gfCNCPoint3[7270] = {X 314.6892, Y 8.8093, Z -3.8333, A 0.000, B 0.000, C 0.000 }
gfCNCPoint3[7271] = {X 315.3732, Y 9.4933, Z -3.8333, A 0.000, B 0.000, C 0.000 }
gfCNCPoint3[7272] = {X 315.8879, Y 10.3124, Z -3.8333, A 0.000, B 0.000, C 0.000 }
gfCNCPoint3[7273] = {X 316.2074, Y 11.2255, Z -3.8333, A 0.000, B 0.000, C 0.000 }
gfCNCPoint3[7274] = {X 316.3157, Y 12.1868, Z -3.8333, A 0.000, B 0.000, C 0.000 }
gfCNCPoint3[7275] = {X 316.3157, Y 12.9781, Z -3.8333, A 0.000, B 0.000, C 0.000 }
gfCNCPoint3[7276] = {X 316.2144, Y 13.9082, Z -3.8333, A 0.000, B 0.000, C 0.000 }
gfCNCPoint3[7277] = {X 315.9152, Y 14.7946, Z -3.8333, A 0.000, B 0.000, C 0.000 }
gfCNCPoint3[7278] = {X 315.4322, Y 15.5958, Z -3.8333, A 0.000, B 0.000, C 0.000 }
gfCNCPoint3[7279] = {X 314.7880, Y 16.2743, Z -3.8333, A 0.000, B 0.000, C 0.000 }
gfCNCPoint3[7280] = {X 314.7878, Y 40.9123, Z -3.8333, A 0.000, B 0.000, C 0.000 }
gfCNCPoint3[7281] = {X 315.4264, Y 41.5834, Z -3.8333, A 0.000, B 0.000, C 0.000 }
gfCNCPoint3[7282] = {X 315.9072, Y 42.3751, Z -3.8333, A 0.000, B 0.000, C 0.000 }
gfCNCPoint3[7283] = {X 316.2082, Y 43.2512, Z -3.8333, A 0.000, B 0.000, C 0.000 }
gfCNCPoint3[7284] = {X 316.3156, Y 44.1713, Z -3.8333, A 0.000, B 0.000, C 0.000 }
gfCNCPoint3[7285] = {X 316.3157, Y 45.0000, Z -3.8333, A 0.000, B 0.000, C 0.000 }
gfCNCPoint3[7286] = {X 316.2074, Y 45.9613, Z -3.8333, A 0.000, B 0.000, C 0.000 }
gfCNCPoint3[7287] = {X 315.8879, Y 46.8744, Z -3.8333, A 0.000, B 0.000, C 0.000 }
gfCNCPoint3[7288] = {X 315.3732, Y 47.6935, Z -3.8333, A 0.000, B 0.000, C 0.000 }
gfCNCPoint3[7289] = {X 314.6892, Y 48.3775, Z -3.8333, A 0.000, B 0.000, C 0.000 }
gfCNCPoint3[7290] = {X 313.8701, Y 48.8922, Z -3.8333, A 0.000, B 0.000, C 0.000 }
gfCNCPoint3[7291] = {X 312.9570, Y 49.2117, Z -3.8333, A 0.000, B 0.000, C 0.000 }
gfCNCPoint3[7292] = {X 311.9957, Y 49.3200, Z -3.8333, A 0.000, B 0.000, C 0.000 }
gfCNCPoint3[7293] = {X 305.5523, Y 49.3200, Z -3.8333, A 0.000, B 0.000, C 0.000 }
gfCNCPoint3[7294] = {X 304.5958, Y 49.2128, Z -3.8333, A 0.000, B 0.000, C 0.000 }
gfCNCPoint3[7295] = {X 303.6868, Y 48.8965, Z -3.8333, A 0.000, B 0.000, C 0.000 }
gfCNCPoint3[7296] = {X 302.8704, Y 48.3868, Z -3.8333, A 0.000, B 0.000, C 0.000 }
gfCNCPoint3[7297] = {X 302.1872, Y 47.7090, Z -3.8333, A 0.000, B 0.000, C 0.000 }
gfCNCPoint3[7298] = {X 301.6709, Y 46.8967, Z -3.8333, A 0.000, B 0.000, C 0.000 }
gfCNCPoint3[7299] = {X 301.3473, Y 45.9903, Z -3.8333, A 0.000, B 0.000, C 0.000 }
gfCNCPoint3[7300] = {X 301.2324, Y 45.0348, Z -3.8333, A 0.000, B 0.000, C 0.000 }
gfCNCPoint3[7301] = {X 301.2323, Y 44.2012, Z -3.8333, A 0.000, B 0.000, C 0.000 }
gfCNCPoint3[7302] = {X 301.3501, Y 43.2651, Z -3.8333, A 0.000, B 0.000, C 0.000 }
gfCNCPoint3[7303] = {X 301.6534, Y 42.3717, Z -3.8333, A 0.000, B 0.000, C 0.000 }
gfCNCPoint3[7304] = {X 302.1298, Y 41.5574, Z -3.8333, A 0.000, B 0.000, C 0.000 }
gfCNCPoint3[7305] = {X 302.7601, Y 40.8554, Z -3.8333, A 0.000, B 0.000, C 0.000 }
gfCNCPoint3[7306] = {X 302.7601, Y 34.0343, Z -3.8333, A 0.000, B 0.000, C 0.000 }
gfCNCPoint3[7307] = {X 293.8542, Y 34.0343, Z -3.8333, A 0.000, B 0.000, C 0.000 }
gfCNCPoint3[7308] = {X 293.8534, Y 40.9025, Z -3.8333, A 0.000, B 0.000, C 0.000 }
gfCNCPoint3[7309] = {X 294.4924, Y 41.5865, Z -3.8333, A 0.000, B 0.000, C 0.000 }
gfCNCPoint3[7310] = {X 294.9731, Y 42.3897, Z -3.8333, A 0.000, B 0.000, C 0.000 }
gfCNCPoint3[7311] = {X 295.2739, Y 43.2762, Z -3.8333, A 0.000, B 0.000, C 0.000 }
gfCNCPoint3[7312] = {X 295.3811, Y 44.2061, Z -3.8333, A 0.000, B 0.000, C 0.000 }
gfCNCPoint3[7313] = {X 295.3811, Y 45.0000, Z -3.8333, A 0.000, B 0.000, C 0.000 }
gfCNCPoint3[7314] = {X 295.2728, Y 45.9613, Z -3.8333, A 0.000, B 0.000, C 0.000 }
gfCNCPoint3[7315] = {X 294.9533, Y 46.8744, Z -3.8333, A 0.000, B 0.000, C 0.000 }
gfCNCPoint3[7316] = {X 294.4386, Y 47.6935, Z -3.8333, A 0.000, B 0.000, C 0.000 }
gfCNCPoint3[7317] = {X 293.7546, Y 48.3775, Z -3.8333, A 0.000, B 0.000, C 0.000 }
gfCNCPoint3[7318] = {X 292.9355, Y 48.8922, Z -3.8333, A 0.000, B 0.000, C 0.000 }
gfCNCPoint3[7319] = {X 292.0224, Y 49.2117, Z -3.8333, A 0.000, B 0.000, C 0.000 }
gfCNCPoint3[7320] = {X 291.0611, Y 49.3200, Z -3.8333, A 0.000, B 0.000, C 0.000 }
gfCNCPoint3[7321] = {X 284.6177, Y 49.3200, Z -3.8333, A 0.000, B 0.000, C 0.000 }
gfCNCPoint3[7322] = {X 283.6613, Y 49.2128, Z -3.8333, A 0.000, B 0.000, C 0.000 }
gfCNCPoint3[7323] = {X 282.7524, Y 48.8965, Z -3.8333, A 0.000, B 0.000, C 0.000 }
gfCNCPoint3[7324] = {X 281.9360, Y 48.3869, Z -3.8333, A 0.000, B 0.000, C 0.000 }
gfCNCPoint3[7325] = {X 281.2527, Y 47.7092, Z -3.8333, A 0.000, B 0.000, C 0.000 }
gfCNCPoint3[7326] = {X 280.7365, Y 46.8970, Z -3.8333, A 0.000, B 0.000, C 0.000 }
gfCNCPoint3[7327] = {X 280.4128, Y 45.9907, Z -3.8333, A 0.000, B 0.000, C 0.000 }
gfCNCPoint3[7328] = {X 280.2978, Y 45.0352, Z -3.8333, A 0.000, B 0.000, C 0.000 }
gfCNCPoint3[7329] = {X 280.2977, Y 44.2072, Z -3.8333, A 0.000, B 0.000, C 0.000 }
gfCNCPoint3[7330] = {X 280.4027, Y 43.2782, Z -3.8333, A 0.000, B 0.000, C 0.000 }
gfCNCPoint3[7331] = {X 280.7029, Y 42.3928, Z -3.8333, A 0.000, B 0.000, C 0.000 }
gfCNCPoint3[7332] = {X 281.1846, Y 41.5915, Z -3.8333, A 0.000, B 0.000, C 0.000 }
gfCNCPoint3[7333] = {X 281.8256, Y 40.9110, Z -3.8333, A 0.000, B 0.000, C 0.000 }
gfCNCPoint3[7334] = {X 281.8254, Y 28.5926, Z -3.8333, A 0.000, B 0.000, C 0.000 }
gfCNCPoint3[7335] = {X 277.8254, Y 28.5927, Z -3.8333, A 0.000, B 0.000, C 0.000 }
gfCNCPoint3[7336] = {X 281.9054, Y 28.5926, Z -3.8333, A 0.000, B 0.000, C 0.000 }
gfCNCPoint3[7337] = {X 281.9052, Y 16.2369, Z -3.8333, A 0.000, B 0.000, C 0.000 }
gfCNCPoint3[7338] = {X 281.2671, Y 15.5764, Z -3.8333, A 0.000, B 0.000, C 0.000 }
gfCNCPoint3[7339] = {X 280.7863, Y 14.7940, Z -3.8333, A 0.000, B 0.000, C 0.000 }
gfCNCPoint3[7340] = {X 280.4851, Y 13.9265, Z -3.8333, A 0.000, B 0.000, C 0.000 }
gfCNCPoint3[7341] = {X 280.3778, Y 13.0144, Z -3.8333, A 0.000, B 0.000, C 0.000 }
gfCNCPoint3[7342] = {X 280.3777, Y 12.1868, Z -3.8333, A 0.000, B 0.000, C 0.000 }
gfCNCPoint3[7343] = {X 280.4840, Y 11.2433, Z -3.8333, A 0.000, B 0.000, C 0.000 }
gfCNCPoint3[7344] = {X 280.7976, Y 10.3472, Z -3.8333, A 0.000, B 0.000, C 0.000 }
gfCNCPoint3[7345] = {X 281.3027, Y 9.5432, Z -3.8333, A 0.000, B 0.000, C 0.000 }
gfCNCPoint3[7346] = {X 281.9741, Y 8.8719, Z -3.8333, A 0.000, B 0.000, C 0.000 }
gfCNCPoint3[7347] = {X 282.7780, Y 8.3667, Z -3.8333, A 0.000, B 0.000, C 0.000 }
gfCNCPoint3[7348] = {X 283.6742, Y 8.0531, Z -3.8333, A 0.000, B 0.000, C 0.000 }
gfCNCPoint3[7349] = {X 284.6177, Y 7.9468, Z -3.8333, A 0.000, B 0.000, C 0.000 }
gfCNCPoint3[7350] = {X 291.0611, Y 7.9468, Z -3.8333, A 0.000, B 0.000, C 0.000 }
gfCNCPoint3[7351] = {X 292.0046, Y 8.0531, Z -3.8333, A 0.000, B 0.000, C 0.000 }
gfCNCPoint3[7352] = {X 292.9008, Y 8.3667, Z -3.8333, A 0.000, B 0.000, C 0.000 }
gfCNCPoint3[7353] = {X 293.7047, Y 8.8718, Z -3.8333, A 0.000, B 0.000, C 0.000 }
gfCNCPoint3[7354] = {X 294.3761, Y 9.5432, Z -3.8333, A 0.000, B 0.000, C 0.000 }
gfCNCPoint3[7355] = {X 294.8812, Y 10.3471, Z -3.8333, A 0.000, B 0.000, C 0.000 }
gfCNCPoint3[7356] = {X 295.1948, Y 11.2433, Z -3.8333, A 0.000, B 0.000, C 0.000 }
gfCNCPoint3[7357] = {X 295.3011, Y 12.1868, Z -3.8333, A 0.000, B 0.000, C 0.000 }
gfCNCPoint3[7358] = {X 295.3011, Y 12.9781, Z -3.8333, A 0.000, B 0.000, C 0.000 }
gfCNCPoint3[7359] = {X 295.1996, Y 13.8999, Z -3.8333, A 0.000, B 0.000, C 0.000 }
gfCNCPoint3[7360] = {X 294.9001, Y 14.7776, Z -3.8333, A 0.000, B 0.000, C 0.000 }
gfCNCPoint3[7361] = {X 294.4170, Y 15.5691, Z -3.8333, A 0.000, B 0.000, C 0.000 }
gfCNCPoint3[7362] = {X 293.7733, Y 16.2367, Z -3.8333, A 0.000, B 0.000, C 0.000 }
gfCNCPoint3[7363] = {X 293.7745, Y 22.2765, Z -3.8333, A 0.000, B 0.000, C 0.000 }
gfCNCPoint3[7364] = {X 302.8393, Y 22.2765, Z -3.8333, A 0.000, B 0.000, C 0.000 }
gfCNCPoint3[7365] = {X 302.8443, Y 16.2406, Z -3.8333, A 0.000, B 0.000, C 0.000 }
gfCNCPoint3[7366] = {X 302.2046, Y 15.5801, Z -3.8333, A 0.000, B 0.000, C 0.000 }
gfCNCPoint3[7367] = {X 301.7224, Y 14.7973, Z -3.8333, A 0.000, B 0.000, C 0.000 }
gfCNCPoint3[7368] = {X 301.4203, Y 13.9289, Z -3.8333, A 0.000, B 0.000, C 0.000 }
gfCNCPoint3[7369] = {X 301.3124, Y 13.0158, Z -3.8333, A 0.000, B 0.000, C 0.000 }
gfCNCPoint3[7370] = {X 301.3123, Y 12.1868, Z -3.8333, A 0.000, B 0.000, C 0.000 }
gfCNCPoint3[7371] = {X 301.4186, Y 11.2433, Z -3.8333, A 0.000, B 0.000, C 0.000 }
gfCNCPoint3[7372] = {X 301.7321, Y 10.3471, Z -3.8333, A 0.000, B 0.000, C 0.000 }
gfCNCPoint3[7373] = {X 302.2373, Y 9.5432, Z -3.8333, A 0.000, B 0.000, C 0.000 }
gfCNCPoint3[7374] = {X 302.9087, Y 8.8718, Z -3.8333, A 0.000, B 0.000, C 0.000 }
gfCNCPoint3[7375] = {X 303.7126, Y 8.3667, Z -3.8333, A 0.000, B 0.000, C 0.000 }
gfCNCPoint3[7376] = {X 304.6088, Y 8.0531, Z -3.8333, A 0.000, B 0.000, C 0.000 }
gfCNCPoint3[7377] = {X 305.5523, Y 7.9468, Z -3.8333, A 0.000, B 0.000, C 0.000 }
gfCNCPoint3[7378] = {X 311.9957, Y 7.9468, Z -3.8333, A 0.000, B 0.000, C 0.000 }
gfCNCPoint3[7379] = {X 312.9392, Y 8.0531, Z -3.8333, A 0.000, B 0.000, C 0.000 }
gfCNCPoint3[7380] = {X 313.8354, Y 8.3667, Z -3.8333, A 0.000, B 0.000, C 0.000 }
gfCNCPoint3[7381] = {X 314.6393, Y 8.8718, Z -3.8333, A 0.000, B 0.000, C 0.000 }
gfCNCPoint3[7382] = {X 315.3107, Y 9.5432, Z -3.8333, A 0.000, B 0.000, C 0.000 }
gfCNCPoint3[7383] = {X 315.8158, Y 10.3471, Z -3.8333, A 0.000, B 0.000, C 0.000 }
gfCNCPoint3[7384] = {X 316.1294, Y 11.2433, Z -3.8333, A 0.000, B 0.000, C 0.000 }
gfCNCPoint3[7385] = {X 316.2357, Y 12.1868, Z -3.8333, A 0.000, B 0.000, C 0.000 }
gfCNCPoint3[7386] = {X 316.2357, Y 12.9781, Z -3.8333, A 0.000, B 0.000, C 0.000 }
gfCNCPoint3[7387] = {X 316.1343, Y 13.9000, Z -3.8333, A 0.000, B 0.000, C 0.000 }
gfCNCPoint3[7388] = {X 315.8348, Y 14.7777, Z -3.8333, A 0.000, B 0.000, C 0.000 }
gfCNCPoint3[7389] = {X 315.3517, Y 15.5693, Z -3.8333, A 0.000, B 0.000, C 0.000 }
gfCNCPoint3[7390] = {X 314.7080, Y 16.2370, Z -3.8333, A 0.000, B 0.000, C 0.000 }
gfCNCPoint3[7391] = {X 314.7078, Y 40.9508, Z -3.8333, A 0.000, B 0.000, C 0.000 }
gfCNCPoint3[7392] = {X 314.7361, Y 40.9734, Z -3.8333, A 0.000, B 0.000, C 0.000 }
gfCNCPoint3[7393] = {X 315.3629, Y 41.6320, Z -3.8333, A 0.000, B 0.000, C 0.000 }
gfCNCPoint3[7394] = {X 315.8348, Y 42.4091, Z -3.8333, A 0.000, B 0.000, C 0.000 }
gfCNCPoint3[7395] = {X 316.1302, Y 43.2689, Z -3.8333, A 0.000, B 0.000, C 0.000 }
gfCNCPoint3[7396] = {X 316.2356, Y 44.1720, Z -3.8333, A 0.000, B 0.000, C 0.000 }
gfCNCPoint3[7397] = {X 316.2357, Y 45.0000, Z -3.8333, A 0.000, B 0.000, C 0.000 }
gfCNCPoint3[7398] = {X 316.1294, Y 45.9435, Z -3.8333, A 0.000, B 0.000, C 0.000 }
gfCNCPoint3[7399] = {X 315.8158, Y 46.8397, Z -3.8333, A 0.000, B 0.000, C 0.000 }
gfCNCPoint3[7400] = {X 315.3107, Y 47.6436, Z -3.8333, A 0.000, B 0.000, C 0.000 }
gfCNCPoint3[7401] = {X 314.6393, Y 48.3150, Z -3.8333, A 0.000, B 0.000, C 0.000 }
gfCNCPoint3[7402] = {X 313.8354, Y 48.8201, Z -3.8333, A 0.000, B 0.000, C 0.000 }
gfCNCPoint3[7403] = {X 312.9392, Y 49.1337, Z -3.8333, A 0.000, B 0.000, C 0.000 }
gfCNCPoint3[7404] = {X 311.9957, Y 49.2400, Z -3.8333, A 0.000, B 0.000, C 0.000 }
gfCNCPoint3[7405] = {X 305.5523, Y 49.2400, Z -3.8333, A 0.000, B 0.000, C 0.000 }
gfCNCPoint3[7406] = {X 304.6135, Y 49.1348, Z -3.8333, A 0.000, B 0.000, C 0.000 }
gfCNCPoint3[7407] = {X 303.7214, Y 48.8243, Z -3.8333, A 0.000, B 0.000, C 0.000 }
gfCNCPoint3[7408] = {X 302.9201, Y 48.3241, Z -3.8333, A 0.000, B 0.000, C 0.000 }
gfCNCPoint3[7409] = {X 302.2495, Y 47.6588, Z -3.8333, A 0.000, B 0.000, C 0.000 }
gfCNCPoint3[7410] = {X 301.7428, Y 46.8616, Z -3.8333, A 0.000, B 0.000, C 0.000 }
gfCNCPoint3[7411] = {X 301.4252, Y 45.9720, Z -3.8333, A 0.000, B 0.000, C 0.000 }
gfCNCPoint3[7412] = {X 301.3124, Y 45.0341, Z -3.8333, A 0.000, B 0.000, C 0.000 }
gfCNCPoint3[7413] = {X 301.3123, Y 44.2031, Z -3.8333, A 0.000, B 0.000, C 0.000 }
gfCNCPoint3[7414] = {X 301.4301, Y 43.2745, Z -3.8333, A 0.000, B 0.000, C 0.000 }
gfCNCPoint3[7415] = {X 301.7335, Y 42.3890, Z -3.8333, A 0.000, B 0.000, C 0.000 }
gfCNCPoint3[7416] = {X 302.2101, Y 41.5833, Z -3.8333, A 0.000, B 0.000, C 0.000 }
gfCNCPoint3[7417] = {X 302.8401, Y 40.8909, Z -3.8333, A 0.000, B 0.000, C 0.000 }
gfCNCPoint3[7418] = {X 302.8401, Y 33.9543, Z -3.8333, A 0.000, B 0.000, C 0.000 }
gfCNCPoint3[7419] = {X 293.7742, Y 33.9543, Z -3.8333, A 0.000, B 0.000, C 0.000 }
gfCNCPoint3[7420] = {X 293.7734, Y 40.9393, Z -3.8333, A 0.000, B 0.000, C 0.000 }
gfCNCPoint3[7421] = {X 294.4120, Y 41.6128, Z -3.8333, A 0.000, B 0.000, C 0.000 }
gfCNCPoint3[7422] = {X 294.8928, Y 42.4068, Z -3.8333, A 0.000, B 0.000, C 0.000 }
gfCNCPoint3[7423] = {X 295.1938, Y 43.2848, Z -3.8333, A 0.000, B 0.000, C 0.000 }
gfCNCPoint3[7424] = {X 295.3011, Y 44.2068, Z -3.8333, A 0.000, B 0.000, C 0.000 }
gfCNCPoint3[7425] = {X 295.3011, Y 45.0000, Z -3.8333, A 0.000, B 0.000, C 0.000 }
gfCNCPoint3[7426] = {X 295.1948, Y 45.9435, Z -3.8333, A 0.000, B 0.000, C 0.000 }
gfCNCPoint3[7427] = {X 294.8812, Y 46.8397, Z -3.8333, A 0.000, B 0.000, C 0.000 }
gfCNCPoint3[7428] = {X 294.3761, Y 47.6436, Z -3.8333, A 0.000, B 0.000, C 0.000 }
gfCNCPoint3[7429] = {X 293.7047, Y 48.3150, Z -3.8333, A 0.000, B 0.000, C 0.000 }
gfCNCPoint3[7430] = {X 292.9008, Y 48.8201, Z -3.8333, A 0.000, B 0.000, C 0.000 }
gfCNCPoint3[7431] = {X 292.0046, Y 49.1337, Z -3.8333, A 0.000, B 0.000, C 0.000 }
gfCNCPoint3[7432] = {X 291.0611, Y 49.2400, Z -3.8333, A 0.000, B 0.000, C 0.000 }
gfCNCPoint3[7433] = {X 284.6177, Y 49.2400, Z -3.8333, A 0.000, B 0.000, C 0.000 }
gfCNCPoint3[7434] = {X 283.6790, Y 49.1348, Z -3.8333, A 0.000, B 0.000, C 0.000 }
gfCNCPoint3[7435] = {X 282.7869, Y 48.8244, Z -3.8333, A 0.000, B 0.000, C 0.000 }
gfCNCPoint3[7436] = {X 281.9857, Y 48.3242, Z -3.8333, A 0.000, B 0.000, C 0.000 }
gfCNCPoint3[7437] = {X 281.3150, Y 47.6590, Z -3.8333, A 0.000, B 0.000, C 0.000 }
gfCNCPoint3[7438] = {X 280.8083, Y 46.8619, Z -3.8333, A 0.000, B 0.000, C 0.000 }
gfCNCPoint3[7439] = {X 280.4907, Y 45.9723, Z -3.8333, A 0.000, B 0.000, C 0.000 }
gfCNCPoint3[7440] = {X 280.3778, Y 45.0345, Z -3.8333, A 0.000, B 0.000, C 0.000 }
gfCNCPoint3[7441] = {X 280.3777, Y 44.2076, Z -3.8333, A 0.000, B 0.000, C 0.000 }
gfCNCPoint3[7442] = {X 280.4828, Y 43.2867, Z -3.8333, A 0.000, B 0.000, C 0.000 }
gfCNCPoint3[7443] = {X 280.7832, Y 42.4098, Z -3.8333, A 0.000, B 0.000, C 0.000 }
gfCNCPoint3[7444] = {X 281.2650, Y 41.6180, Z -3.8333, A 0.000, B 0.000, C 0.000 }
gfCNCPoint3[7445] = {X 281.9056, Y 40.9481, Z -3.8333, A 0.000, B 0.000, C 0.000 }
gfCNCPoint3[7446] = {X 281.9054, Y 28.5926, Z -3.8333, A 0.000, B 0.000, C 0.000 }
gfCNCPoint3[7447] = {X 277.9054, Y 28.5927, Z -3.8333, A 0.000, B 0.000, C 0.000 }
gfCNCPoint3[7448] = {X 281.9854, Y 28.5926, Z -3.8333, A 0.000, B 0.000, C 0.000 }
gfCNCPoint3[7449] = {X 281.9852, Y 16.1992, Z -3.8333, A 0.000, B 0.000, C 0.000 }
gfCNCPoint3[7450] = {X 281.3476, Y 15.5495, Z -3.8333, A 0.000, B 0.000, C 0.000 }
gfCNCPoint3[7451] = {X 280.8666, Y 14.7766, Z -3.8333, A 0.000, B 0.000, C 0.000 }
gfCNCPoint3[7452] = {X 280.5652, Y 13.9177, Z -3.8333, A 0.000, B 0.000, C 0.000 }
gfCNCPoint3[7453] = {X 280.4578, Y 13.0137, Z -3.8333, A 0.000, B 0.000, C 0.000 }
gfCNCPoint3[7454] = {X 280.4577, Y 12.1868, Z -3.8333, A 0.000, B 0.000, C 0.000 }
gfCNCPoint3[7455] = {X 280.5620, Y 11.2611, Z -3.8333, A 0.000, B 0.000, C 0.000 }
gfCNCPoint3[7456] = {X 280.8696, Y 10.3819, Z -3.8333, A 0.000, B 0.000, C 0.000 }
gfCNCPoint3[7457] = {X 281.3652, Y 9.5931, Z -3.8333, A 0.000, B 0.000, C 0.000 }
gfCNCPoint3[7458] = {X 282.0240, Y 8.9344, Z -3.8333, A 0.000, B 0.000, C 0.000 }
gfCNCPoint3[7459] = {X 282.8127, Y 8.4388, Z -3.8333, A 0.000, B 0.000, C 0.000 }
gfCNCPoint3[7460] = {X 283.6920, Y 8.1311, Z -3.8333, A 0.000, B 0.000, C 0.000 }
gfCNCPoint3[7461] = {X 284.6177, Y 8.0268, Z -3.8333, A 0.000, B 0.000, C 0.000 }
gfCNCPoint3[7462] = {X 291.0611, Y 8.0268, Z -3.8333, A 0.000, B 0.000, C 0.000 }
gfCNCPoint3[7463] = {X 291.9868, Y 8.1311, Z -3.8333, A 0.000, B 0.000, C 0.000 }
gfCNCPoint3[7464] = {X 292.8661, Y 8.4388, Z -3.8333, A 0.000, B 0.000, C 0.000 }
gfCNCPoint3[7465] = {X 293.6549, Y 8.9344, Z -3.8333, A 0.000, B 0.000, C 0.000 }
gfCNCPoint3[7466] = {X 294.3136, Y 9.5931, Z -3.8333, A 0.000, B 0.000, C 0.000 }
gfCNCPoint3[7467] = {X 294.8092, Y 10.3819, Z -3.8333, A 0.000, B 0.000, C 0.000 }
gfCNCPoint3[7468] = {X 295.1168, Y 11.2611, Z -3.8333, A 0.000, B 0.000, C 0.000 }
gfCNCPoint3[7469] = {X 295.2211, Y 12.1868, Z -3.8333, A 0.000, B 0.000, C 0.000 }
gfCNCPoint3[7470] = {X 295.2211, Y 12.9781, Z -3.8333, A 0.000, B 0.000, C 0.000 }
gfCNCPoint3[7471] = {X 295.1254, Y 13.8652, Z -3.8333, A 0.000, B 0.000, C 0.000 }
gfCNCPoint3[7472] = {X 294.8428, Y 14.7115, Z -3.8333, A 0.000, B 0.000, C 0.000 }
gfCNCPoint3[7473] = {X 294.3862, Y 15.4780, Z -3.8333, A 0.000, B 0.000, C 0.000 }
gfCNCPoint3[7474] = {X 293.7766, Y 16.1295, Z -3.8333, A 0.000, B 0.000, C 0.000 }
gfCNCPoint3[7475] = {X 293.6933, Y 16.1994, Z -3.8333, A 0.000, B 0.000, C 0.000 }
gfCNCPoint3[7476] = {X 293.6945, Y 22.3566, Z -3.8333, A 0.000, B 0.000, C 0.000 }
gfCNCPoint3[7477] = {X 302.9192, Y 22.3565, Z -3.8333, A 0.000, B 0.000, C 0.000 }
gfCNCPoint3[7478] = {X 302.9243, Y 16.2028, Z -3.8333, A 0.000, B 0.000, C 0.000 }
gfCNCPoint3[7479] = {X 302.2851, Y 15.5532, Z -3.8333, A 0.000, B 0.000, C 0.000 }
gfCNCPoint3[7480] = {X 301.8027, Y 14.7799, Z -3.8333, A 0.000, B 0.000, C 0.000 }
gfCNCPoint3[7481] = {X 301.5003, Y 13.9201, Z -3.8333, A 0.000, B 0.000, C 0.000 }
gfCNCPoint3[7482] = {X 301.3924, Y 13.0151, Z -3.8333, A 0.000, B 0.000, C 0.000 }
gfCNCPoint3[7483] = {X 301.3923, Y 12.1868, Z -3.8333, A 0.000, B 0.000, C 0.000 }
gfCNCPoint3[7484] = {X 301.4966, Y 11.2611, Z -3.8333, A 0.000, B 0.000, C 0.000 }
gfCNCPoint3[7485] = {X 301.8042, Y 10.3819, Z -3.8333, A 0.000, B 0.000, C 0.000 }
gfCNCPoint3[7486] = {X 302.2998, Y 9.5931, Z -3.8333, A 0.000, B 0.000, C 0.000 }
gfCNCPoint3[7487] = {X 302.9585, Y 8.9344, Z -3.8333, A 0.000, B 0.000, C 0.000 }
gfCNCPoint3[7488] = {X 303.7473, Y 8.4388, Z -3.8333, A 0.000, B 0.000, C 0.000 }
gfCNCPoint3[7489] = {X 304.6266, Y 8.1311, Z -3.8333, A 0.000, B 0.000, C 0.000 }
gfCNCPoint3[7490] = {X 305.5523, Y 8.0268, Z -3.8333, A 0.000, B 0.000, C 0.000 }
gfCNCPoint3[7491] = {X 311.9957, Y 8.0268, Z -3.8333, A 0.000, B 0.000, C 0.000 }
gfCNCPoint3[7492] = {X 312.9214, Y 8.1311, Z -3.8333, A 0.000, B 0.000, C 0.000 }
gfCNCPoint3[7493] = {X 313.8007, Y 8.4388, Z -3.8333, A 0.000, B 0.000, C 0.000 }
gfCNCPoint3[7494] = {X 314.5894, Y 8.9344, Z -3.8333, A 0.000, B 0.000, C 0.000 }
gfCNCPoint3[7495] = {X 315.2481, Y 9.5931, Z -3.8333, A 0.000, B 0.000, C 0.000 }
gfCNCPoint3[7496] = {X 315.7438, Y 10.3819, Z -3.8333, A 0.000, B 0.000, C 0.000 }
gfCNCPoint3[7497] = {X 316.0514, Y 11.2611, Z -3.8333, A 0.000, B 0.000, C 0.000 }
gfCNCPoint3[7498] = {X 316.1557, Y 12.1868, Z -3.8333, A 0.000, B 0.000, C 0.000 }
gfCNCPoint3[7499] = {X 316.1557, Y 12.9781, Z -3.8333, A 0.000, B 0.000, C 0.000 }
gfCNCPoint3[7500] = {X 316.0542, Y 13.8916, Z -3.8333, A 0.000, B 0.000, C 0.000 }
gfCNCPoint3[7501] = {X 315.7545, Y 14.7604, Z -3.8333, A 0.000, B 0.000, C 0.000 }
gfCNCPoint3[7502] = {X 315.2715, Y 15.5422, Z -3.8333, A 0.000, B 0.000, C 0.000 }
gfCNCPoint3[7503] = {X 314.6285, Y 16.1989, Z -3.8333, A 0.000, B 0.000, C 0.000 }
gfCNCPoint3[7504] = {X 314.6278, Y 40.9894, Z -3.8333, A 0.000, B 0.000, C 0.000 }
gfCNCPoint3[7505] = {X 314.6834, Y 41.0336, Z -3.8333, A 0.000, B 0.000, C 0.000 }
gfCNCPoint3[7506] = {X 315.2987, Y 41.6798, Z -3.8333, A 0.000, B 0.000, C 0.000 }
gfCNCPoint3[7507] = {X 315.7621, Y 42.4424, Z -3.8333, A 0.000, B 0.000, C 0.000 }
gfCNCPoint3[7508] = {X 316.0522, Y 43.2863, Z -3.8333, A 0.000, B 0.000, C 0.000 }
gfCNCPoint3[7509] = {X 316.1556, Y 44.1727, Z -3.8333, A 0.000, B 0.000, C 0.000 }
gfCNCPoint3[7510] = {X 316.1557, Y 45.0000, Z -3.8333, A 0.000, B 0.000, C 0.000 }
gfCNCPoint3[7511] = {X 316.0514, Y 45.9257, Z -3.8333, A 0.000, B 0.000, C 0.000 }
gfCNCPoint3[7512] = {X 315.7438, Y 46.8050, Z -3.8333, A 0.000, B 0.000, C 0.000 }
gfCNCPoint3[7513] = {X 315.2481, Y 47.5937, Z -3.8333, A 0.000, B 0.000, C 0.000 }
gfCNCPoint3[7514] = {X 314.5894, Y 48.2524, Z -3.8333, A 0.000, B 0.000, C 0.000 }
gfCNCPoint3[7515] = {X 313.8007, Y 48.7480, Z -3.8333, A 0.000, B 0.000, C 0.000 }
gfCNCPoint3[7516] = {X 312.9214, Y 49.0557, Z -3.8333, A 0.000, B 0.000, C 0.000 }
gfCNCPoint3[7517] = {X 311.9957, Y 49.1600, Z -3.8333, A 0.000, B 0.000, C 0.000 }
gfCNCPoint3[7518] = {X 305.5523, Y 49.1600, Z -3.8333, A 0.000, B 0.000, C 0.000 }
gfCNCPoint3[7519] = {X 304.6312, Y 49.0568, Z -3.8333, A 0.000, B 0.000, C 0.000 }
gfCNCPoint3[7520] = {X 303.7559, Y 48.7522, Z -3.8333, A 0.000, B 0.000, C 0.000 }
gfCNCPoint3[7521] = {X 302.9698, Y 48.2613, Z -3.8333, A 0.000, B 0.000, C 0.000 }
gfCNCPoint3[7522] = {X 302.3118, Y 47.6087, Z -3.8333, A 0.000, B 0.000, C 0.000 }
gfCNCPoint3[7523] = {X 301.8147, Y 46.8265, Z -3.8333, A 0.000, B 0.000, C 0.000 }
gfCNCPoint3[7524] = {X 301.5030, Y 45.9537, Z -3.8333, A 0.000, B 0.000, C 0.000 }
gfCNCPoint3[7525] = {X 301.3924, Y 45.0335, Z -3.8333, A 0.000, B 0.000, C 0.000 }
gfCNCPoint3[7526] = {X 301.3923, Y 44.2050, Z -3.8333, A 0.000, B 0.000, C 0.000 }
gfCNCPoint3[7527] = {X 301.5100, Y 43.2839, Z -3.8333, A 0.000, B 0.000, C 0.000 }
gfCNCPoint3[7528] = {X 301.8136, Y 42.4063, Z -3.8333, A 0.000, B 0.000, C 0.000 }
gfCNCPoint3[7529] = {X 302.2904, Y 41.6094, Z -3.8333, A 0.000, B 0.000, C 0.000 }
gfCNCPoint3[7530] = {X 302.9201, Y 40.9268, Z -3.8333, A 0.000, B 0.000, C 0.000 }
gfCNCPoint3[7531] = {X 302.9201, Y 33.8743, Z -3.8333, A 0.000, B 0.000, C 0.000 }
gfCNCPoint3[7532] = {X 293.6942, Y 33.8743, Z -3.8333, A 0.000, B 0.000, C 0.000 }
gfCNCPoint3[7533] = {X 293.6934, Y 40.9764, Z -3.8333, A 0.000, B 0.000, C 0.000 }
gfCNCPoint3[7534] = {X 294.3316, Y 41.6394, Z -3.8333, A 0.000, B 0.000, C 0.000 }
gfCNCPoint3[7535] = {X 294.8125, Y 42.4240, Z -3.8333, A 0.000, B 0.000, C 0.000 }
gfCNCPoint3[7536] = {X 295.1137, Y 43.2935, Z -3.8333, A 0.000, B 0.000, C 0.000 }
gfCNCPoint3[7537] = {X 295.2211, Y 44.2075, Z -3.8333, A 0.000, B 0.000, C 0.000 }
gfCNCPoint3[7538] = {X 295.2211, Y 45.0000, Z -3.8333, A 0.000, B 0.000, C 0.000 }
gfCNCPoint3[7539] = {X 295.1168, Y 45.9257, Z -3.8333, A 0.000, B 0.000, C 0.000 }
gfCNCPoint3[7540] = {X 294.8092, Y 46.8050, Z -3.8333, A 0.000, B 0.000, C 0.000 }
gfCNCPoint3[7541] = {X 294.3136, Y 47.5937, Z -3.8333, A 0.000, B 0.000, C 0.000 }
gfCNCPoint3[7542] = {X 293.6549, Y 48.2524, Z -3.8333, A 0.000, B 0.000, C 0.000 }
gfCNCPoint3[7543] = {X 292.8661, Y 48.7480, Z -3.8333, A 0.000, B 0.000, C 0.000 }
gfCNCPoint3[7544] = {X 291.9868, Y 49.0557, Z -3.8333, A 0.000, B 0.000, C 0.000 }
gfCNCPoint3[7545] = {X 291.0611, Y 49.1600, Z -3.8333, A 0.000, B 0.000, C 0.000 }
gfCNCPoint3[7546] = {X 284.6177, Y 49.1600, Z -3.8333, A 0.000, B 0.000, C 0.000 }
gfCNCPoint3[7547] = {X 283.6967, Y 49.0568, Z -3.8333, A 0.000, B 0.000, C 0.000 }
gfCNCPoint3[7548] = {X 282.8214, Y 48.7522, Z -3.8333, A 0.000, B 0.000, C 0.000 }
gfCNCPoint3[7549] = {X 282.0353, Y 48.2615, Z -3.8333, A 0.000, B 0.000, C 0.000 }
gfCNCPoint3[7550] = {X 281.3774, Y 47.6088, Z -3.8333, A 0.000, B 0.000, C 0.000 }
gfCNCPoint3[7551] = {X 280.8802, Y 46.8267, Z -3.8333, A 0.000, B 0.000, C 0.000 }
gfCNCPoint3[7552] = {X 280.5685, Y 45.9540, Z -3.8333, A 0.000, B 0.000, C 0.000 }
gfCNCPoint3[7553] = {X 280.4578, Y 45.0339, Z -3.8333, A 0.000, B 0.000, C 0.000 }
gfCNCPoint3[7554] = {X 280.4577, Y 44.2080, Z -3.8333, A 0.000, B 0.000, C 0.000 }
gfCNCPoint3[7555] = {X 280.5629, Y 43.2952, Z -3.8333, A 0.000, B 0.000, C 0.000 }
gfCNCPoint3[7556] = {X 280.8636, Y 42.4270, Z -3.8333, A 0.000, B 0.000, C 0.000 }
gfCNCPoint3[7557] = {X 281.3455, Y 41.6447, Z -3.8333, A 0.000, B 0.000, C 0.000 }
gfCNCPoint3[7558] = {X 281.9856, Y 40.9855, Z -3.8333, A 0.000, B 0.000, C 0.000 }
gfCNCPoint3[7559] = {X 281.9854, Y 28.5926, Z -3.8333, A 0.000, B 0.000, C 0.000 }
gfCNCPoint3[7560] = {X 277.9854, Y 28.5927, Z -3.8333, A 0.000, B 0.000, C 0.000 }
gfCNCPoint3[7561] = {X 282.0654, Y 28.5926, Z -3.8333, A 0.000, B 0.000, C 0.000 }
gfCNCPoint3[7562] = {X 282.0652, Y 16.1610, Z -3.8333, A 0.000, B 0.000, C 0.000 }
gfCNCPoint3[7563] = {X 281.4281, Y 15.5222, Z -3.8333, A 0.000, B 0.000, C 0.000 }
gfCNCPoint3[7564] = {X 280.9469, Y 14.7591, Z -3.8333, A 0.000, B 0.000, C 0.000 }
gfCNCPoint3[7565] = {X 280.6453, Y 13.9088, Z -3.8333, A 0.000, B 0.000, C 0.000 }
gfCNCPoint3[7566] = {X 280.5378, Y 13.0130, Z -3.8333, A 0.000, B 0.000, C 0.000 }
gfCNCPoint3[7567] = {X 280.5377, Y 12.1868, Z -3.8333, A 0.000, B 0.000, C 0.000 }
gfCNCPoint3[7568] = {X 280.6400, Y 11.2789, Z -3.8333, A 0.000, B 0.000, C 0.000 }
gfCNCPoint3[7569] = {X 280.9417, Y 10.4166, Z -3.8333, A 0.000, B 0.000, C 0.000 }
gfCNCPoint3[7570] = {X 281.4278, Y 9.6430, Z -3.8333, A 0.000, B 0.000, C 0.000 }
gfCNCPoint3[7571] = {X 282.0738, Y 8.9969, Z -3.8333, A 0.000, B 0.000, C 0.000 }
gfCNCPoint3[7572] = {X 282.8474, Y 8.5109, Z -3.8333, A 0.000, B 0.000, C 0.000 }
gfCNCPoint3[7573] = {X 283.7098, Y 8.2091, Z -3.8333, A 0.000, B 0.000, C 0.000 }
gfCNCPoint3[7574] = {X 284.6177, Y 8.1068, Z -3.8333, A 0.000, B 0.000, C 0.000 }
gfCNCPoint3[7575] = {X 291.0611, Y 8.1068, Z -3.8333, A 0.000, B 0.000, C 0.000 }
gfCNCPoint3[7576] = {X 291.9690, Y 8.2091, Z -3.8333, A 0.000, B 0.000, C 0.000 }
gfCNCPoint3[7577] = {X 292.8314, Y 8.5109, Z -3.8333, A 0.000, B 0.000, C 0.000 }
gfCNCPoint3[7578] = {X 293.6050, Y 8.9969, Z -3.8333, A 0.000, B 0.000, C 0.000 }
gfCNCPoint3[7579] = {X 294.2510, Y 9.6430, Z -3.8333, A 0.000, B 0.000, C 0.000 }
gfCNCPoint3[7580] = {X 294.7371, Y 10.4166, Z -3.8333, A 0.000, B 0.000, C 0.000 }
gfCNCPoint3[7581] = {X 295.0388, Y 11.2789, Z -3.8333, A 0.000, B 0.000, C 0.000 }
gfCNCPoint3[7582] = {X 295.1411, Y 12.1868, Z -3.8333, A 0.000, B 0.000, C 0.000 }
gfCNCPoint3[7583] = {X 295.1411, Y 12.9781, Z -3.8333, A 0.000, B 0.000, C 0.000 }
gfCNCPoint3[7584] = {X 295.0473, Y 13.8481, Z -3.8333, A 0.000, B 0.000, C 0.000 }
gfCNCPoint3[7585] = {X 294.7701, Y 14.6781, Z -3.8333, A 0.000, B 0.000, C 0.000 }
gfCNCPoint3[7586] = {X 294.3222, Y 15.4299, Z -3.8333, A 0.000, B 0.000, C 0.000 }
gfCNCPoint3[7587] = {X 293.7244, Y 16.0689, Z -3.8333, A 0.000, B 0.000, C 0.000 }
gfCNCPoint3[7588] = {X 293.6670, Y 16.1174, Z -3.8333, A 0.000, B 0.000, C 0.000 }
gfCNCPoint3[7589] = {X 293.6087, Y 16.1649, Z -3.8333, A 0.000, B 0.000, C 0.000 }
gfCNCPoint3[7590] = {X 293.6133, Y 16.1995, Z -3.8333, A 0.000, B 0.000, C 0.000 }
gfCNCPoint3[7591] = {X 293.6145, Y 22.4367, Z -3.8333, A 0.000, B 0.000, C 0.000 }
gfCNCPoint3[7592] = {X 293.7676, Y 22.4365, Z -3.8333, A 0.000, B 0.000, C 0.000 }
gfCNCPoint3[7593] = {X 302.9992, Y 22.4365, Z -3.8333, A 0.000, B 0.000, C 0.000 }
gfCNCPoint3[7594] = {X 303.0043, Y 16.1646, Z -3.8333, A 0.000, B 0.000, C 0.000 }
gfCNCPoint3[7595] = {X 302.9460, Y 16.1171, Z -3.8333, A 0.000, B 0.000, C 0.000 }
gfCNCPoint3[7596] = {X 302.8886, Y 16.0686, Z -3.8333, A 0.000, B 0.000, C 0.000 }
gfCNCPoint3[7597] = {X 302.2964, Y 15.4368, Z -3.8333, A 0.000, B 0.000, C 0.000 }
gfCNCPoint3[7598] = {X 301.8508, Y 14.6944, Z -3.8333, A 0.000, B 0.000, C 0.000 }
gfCNCPoint3[7599] = {X 301.5720, Y 13.8746, Z -3.8333, A 0.000, B 0.000, C 0.000 }
gfCNCPoint3[7600] = {X 301.4724, Y 13.0144, Z -3.8333, A 0.000, B 0.000, C 0.000 }
gfCNCPoint3[7601] = {X 301.4723, Y 12.1868, Z -3.8333, A 0.000, B 0.000, C 0.000 }
gfCNCPoint3[7602] = {X 301.5745, Y 11.2789, Z -3.8333, A 0.000, B 0.000, C 0.000 }
gfCNCPoint3[7603] = {X 301.8763, Y 10.4166, Z -3.8333, A 0.000, B 0.000, C 0.000 }
gfCNCPoint3[7604] = {X 302.3624, Y 9.6430, Z -3.8333, A 0.000, B 0.000, C 0.000 }
gfCNCPoint3[7605] = {X 303.0084, Y 8.9969, Z -3.8333, A 0.000, B 0.000, C 0.000 }
gfCNCPoint3[7606] = {X 303.7820, Y 8.5109, Z -3.8333, A 0.000, B 0.000, C 0.000 }
gfCNCPoint3[7607] = {X 304.6444, Y 8.2091, Z -3.8333, A 0.000, B 0.000, C 0.000 }
gfCNCPoint3[7608] = {X 305.5523, Y 8.1068, Z -3.8333, A 0.000, B 0.000, C 0.000 }
gfCNCPoint3[7609] = {X 311.9957, Y 8.1068, Z -3.8333, A 0.000, B 0.000, C 0.000 }
gfCNCPoint3[7610] = {X 312.9036, Y 8.2091, Z -3.8333, A 0.000, B 0.000, C 0.000 }
gfCNCPoint3[7611] = {X 313.7660, Y 8.5109, Z -3.8333, A 0.000, B 0.000, C 0.000 }
gfCNCPoint3[7612] = {X 314.5396, Y 8.9969, Z -3.8333, A 0.000, B 0.000, C 0.000 }
gfCNCPoint3[7613] = {X 315.1856, Y 9.6430, Z -3.8333, A 0.000, B 0.000, C 0.000 }
gfCNCPoint3[7614] = {X 315.6717, Y 10.4166, Z -3.8333, A 0.000, B 0.000, C 0.000 }
gfCNCPoint3[7615] = {X 315.9734, Y 11.2789, Z -3.8333, A 0.000, B 0.000, C 0.000 }
gfCNCPoint3[7616] = {X 316.0757, Y 12.1868, Z -3.8333, A 0.000, B 0.000, C 0.000 }
gfCNCPoint3[7617] = {X 316.0757, Y 12.9781, Z -3.8333, A 0.000, B 0.000, C 0.000 }
gfCNCPoint3[7618] = {X 315.9819, Y 13.8481, Z -3.8333, A 0.000, B 0.000, C 0.000 }
gfCNCPoint3[7619] = {X 315.7047, Y 14.6780, Z -3.8333, A 0.000, B 0.000, C 0.000 }
gfCNCPoint3[7620] = {X 315.2569, Y 15.4298, Z -3.8333, A 0.000, B 0.000, C 0.000 }
gfCNCPoint3[7621] = {X 314.6591, Y 16.0687, Z -3.8333, A 0.000, B 0.000, C 0.000 }
gfCNCPoint3[7622] = {X 314.6045, Y 16.1150, Z -3.8333, A 0.000, B 0.000, C 0.000 }
gfCNCPoint3[7623] = {X 314.5490, Y 16.1603, Z -3.8333, A 0.000, B 0.000, C 0.000 }
gfCNCPoint3[7624] = {X 314.5478, Y 41.0280, Z -3.8333, A 0.000, B 0.000, C 0.000 }
gfCNCPoint3[7625] = {X 314.6336, Y 41.0962, Z -3.8333, A 0.000, B 0.000, C 0.000 }
gfCNCPoint3[7626] = {X 315.2363, Y 41.7299, Z -3.8333, A 0.000, B 0.000, C 0.000 }
gfCNCPoint3[7627] = {X 315.6902, Y 42.4775, Z -3.8333, A 0.000, B 0.000, C 0.000 }
gfCNCPoint3[7628] = {X 315.9743, Y 43.3047, Z -3.8333, A 0.000, B 0.000, C 0.000 }
gfCNCPoint3[7629] = {X 316.0756, Y 44.1734, Z -3.8333, A 0.000, B 0.000, C 0.000 }
gfCNCPoint3[7630] = {X 316.0757, Y 45.0000, Z -3.8333, A 0.000, B 0.000, C 0.000 }
gfCNCPoint3[7631] = {X 315.9734, Y 45.9079, Z -3.8333, A 0.000, B 0.000, C 0.000 }
gfCNCPoint3[7632] = {X 315.6717, Y 46.7702, Z -3.8333, A 0.000, B 0.000, C 0.000 }
gfCNCPoint3[7633] = {X 315.1856, Y 47.5438, Z -3.8333, A 0.000, B 0.000, C 0.000 }
gfCNCPoint3[7634] = {X 314.5396, Y 48.1899, Z -3.8333, A 0.000, B 0.000, C 0.000 }
gfCNCPoint3[7635] = {X 313.7660, Y 48.6760, Z -3.8333, A 0.000, B 0.000, C 0.000 }
gfCNCPoint3[7636] = {X 312.9036, Y 48.9777, Z -3.8333, A 0.000, B 0.000, C 0.000 }
gfCNCPoint3[7637] = {X 311.9957, Y 49.0800, Z -3.8333, A 0.000, B 0.000, C 0.000 }
gfCNCPoint3[7638] = {X 305.5523, Y 49.0800, Z -3.8333, A 0.000, B 0.000, C 0.000 }
gfCNCPoint3[7639] = {X 304.6489, Y 48.9787, Z -3.8333, A 0.000, B 0.000, C 0.000 }
gfCNCPoint3[7640] = {X 303.7905, Y 48.6800, Z -3.8333, A 0.000, B 0.000, C 0.000 }
gfCNCPoint3[7641] = {X 303.0194, Y 48.1986, Z -3.8333, A 0.000, B 0.000, C 0.000 }
gfCNCPoint3[7642] = {X 302.3741, Y 47.5585, Z -3.8333, A 0.000, B 0.000, C 0.000 }
gfCNCPoint3[7643] = {X 301.8865, Y 46.7914, Z -3.8333, A 0.000, B 0.000, C 0.000 }
gfCNCPoint3[7644] = {X 301.5809, Y 45.9353, Z -3.8333, A 0.000, B 0.000, C 0.000 }
gfCNCPoint3[7645] = {X 301.4724, Y 45.0328, Z -3.8333, A 0.000, B 0.000, C 0.000 }
gfCNCPoint3[7646] = {X 301.4723, Y 44.2070, Z -3.8333, A 0.000, B 0.000, C 0.000 }
gfCNCPoint3[7647] = {X 301.5900, Y 43.2934, Z -3.8333, A 0.000, B 0.000, C 0.000 }
gfCNCPoint3[7648] = {X 301.8938, Y 42.4238, Z -3.8333, A 0.000, B 0.000, C 0.000 }
gfCNCPoint3[7649] = {X 302.3707, Y 41.6357, Z -3.8333, A 0.000, B 0.000, C 0.000 }
gfCNCPoint3[7650] = {X 303.0001, Y 40.9632, Z -3.8333, A 0.000, B 0.000, C 0.000 }
gfCNCPoint3[7651] = {X 303.0001, Y 33.7943, Z -3.8333, A 0.000, B 0.000, C 0.000 }
gfCNCPoint3[7652] = {X 293.6143, Y 33.7943, Z -3.8333, A 0.000, B 0.000, C 0.000 }
gfCNCPoint3[7653] = {X 293.6134, Y 41.0141, Z -3.8333, A 0.000, B 0.000, C 0.000 }
gfCNCPoint3[7654] = {X 294.2511, Y 41.6663, Z -3.8333, A 0.000, B 0.000, C 0.000 }
gfCNCPoint3[7655] = {X 294.7322, Y 42.4413, Z -3.8333, A 0.000, B 0.000, C 0.000 }
gfCNCPoint3[7656] = {X 295.0337, Y 43.3023, Z -3.8333, A 0.000, B 0.000, C 0.000 }
gfCNCPoint3[7657] = {X 295.1411, Y 44.2082, Z -3.8333, A 0.000, B 0.000, C 0.000 }
gfCNCPoint3[7658] = {X 295.1411, Y 45.0000, Z -3.8333, A 0.000, B 0.000, C 0.000 }
gfCNCPoint3[7659] = {X 295.0388, Y 45.9079, Z -3.8333, A 0.000, B 0.000, C 0.000 }
gfCNCPoint3[7660] = {X 294.7371, Y 46.7702, Z -3.8333, A 0.000, B 0.000, C 0.000 }
gfCNCPoint3[7661] = {X 294.2510, Y 47.5438, Z -3.8333, A 0.000, B 0.000, C 0.000 }
gfCNCPoint3[7662] = {X 293.6050, Y 48.1899, Z -3.8333, A 0.000, B 0.000, C 0.000 }
gfCNCPoint3[7663] = {X 292.8314, Y 48.6760, Z -3.8333, A 0.000, B 0.000, C 0.000 }
gfCNCPoint3[7664] = {X 291.9690, Y 48.9777, Z -3.8333, A 0.000, B 0.000, C 0.000 }
gfCNCPoint3[7665] = {X 291.0611, Y 49.0800, Z -3.8333, A 0.000, B 0.000, C 0.000 }
gfCNCPoint3[7666] = {X 284.6177, Y 49.0800, Z -3.8333, A 0.000, B 0.000, C 0.000 }
gfCNCPoint3[7667] = {X 283.7144, Y 48.9788, Z -3.8333, A 0.000, B 0.000, C 0.000 }
gfCNCPoint3[7668] = {X 282.8560, Y 48.6801, Z -3.8333, A 0.000, B 0.000, C 0.000 }
gfCNCPoint3[7669] = {X 282.0850, Y 48.1987, Z -3.8333, A 0.000, B 0.000, C 0.000 }
gfCNCPoint3[7670] = {X 281.4397, Y 47.5587, Z -3.8333, A 0.000, B 0.000, C 0.000 }
gfCNCPoint3[7671] = {X 280.9521, Y 46.7916, Z -3.8333, A 0.000, B 0.000, C 0.000 }
gfCNCPoint3[7672] = {X 280.6464, Y 45.9356, Z -3.8333, A 0.000, B 0.000, C 0.000 }
gfCNCPoint3[7673] = {X 280.5378, Y 45.0332, Z -3.8333, A 0.000, B 0.000, C 0.000 }
gfCNCPoint3[7674] = {X 280.5377, Y 44.2085, Z -3.8333, A 0.000, B 0.000, C 0.000 }
gfCNCPoint3[7675] = {X 280.6430, Y 43.3039, Z -3.8333, A 0.000, B 0.000, C 0.000 }
gfCNCPoint3[7676] = {X 280.9439, Y 42.4443, Z -3.8333, A 0.000, B 0.000, C 0.000 }
gfCNCPoint3[7677] = {X 281.4260, Y 41.6717, Z -3.8333, A 0.000, B 0.000, C 0.000 }
gfCNCPoint3[7678] = {X 282.0656, Y 41.0234, Z -3.8333, A 0.000, B 0.000, C 0.000 }
gfCNCPoint3[7679] = {X 282.0654, Y 28.5926, Z -3.8333, A 0.000, B 0.000, C 0.000 }
gfCNCPoint3[7680] = {X 278.0654, Y 28.5927, Z -3.8333, A 0.000, B 0.000, C 0.000 }
gfCNCPoint3[7681] = {X 282.1454, Y 28.5926, Z -3.8333, A 0.000, B 0.000, C 0.000 }
gfCNCPoint3[7682] = {X 282.1452, Y 16.1224, Z -3.8333, A 0.000, B 0.000, C 0.000 }
gfCNCPoint3[7683] = {X 281.5032, Y 15.4880, Z -3.8333, A 0.000, B 0.000, C 0.000 }
gfCNCPoint3[7684] = {X 281.0197, Y 14.7259, Z -3.8333, A 0.000, B 0.000, C 0.000 }
gfCNCPoint3[7685] = {X 280.7195, Y 13.8747, Z -3.8333, A 0.000, B 0.000, C 0.000 }
gfCNCPoint3[7686] = {X 280.6177, Y 12.9779, Z -3.8333, A 0.000, B 0.000, C 0.000 }
gfCNCPoint3[7687] = {X 280.6177, Y 12.1868, Z -3.8333, A 0.000, B 0.000, C 0.000 }
gfCNCPoint3[7688] = {X 280.7180, Y 11.2967, Z -3.8333, A 0.000, B 0.000, C 0.000 }
gfCNCPoint3[7689] = {X 281.0138, Y 10.4513, Z -3.8333, A 0.000, B 0.000, C 0.000 }
gfCNCPoint3[7690] = {X 281.4903, Y 9.6929, Z -3.8333, A 0.000, B 0.000, C 0.000 }
gfCNCPoint3[7691] = {X 282.1237, Y 9.0595, Z -3.8333, A 0.000, B 0.000, C 0.000 }
gfCNCPoint3[7692] = {X 282.8821, Y 8.5829, Z -3.8333, A 0.000, B 0.000, C 0.000 }
gfCNCPoint3[7693] = {X 283.7276, Y 8.2871, Z -3.8333, A 0.000, B 0.000, C 0.000 }
gfCNCPoint3[7694] = {X 284.6177, Y 8.1868, Z -3.8333, A 0.000, B 0.000, C 0.000 }
gfCNCPoint3[7695] = {X 291.0611, Y 8.1868, Z -3.8333, A 0.000, B 0.000, C 0.000 }
gfCNCPoint3[7696] = {X 291.9512, Y 8.2871, Z -3.8333, A 0.000, B 0.000, C 0.000 }
gfCNCPoint3[7697] = {X 292.7967, Y 8.5829, Z -3.8333, A 0.000, B 0.000, C 0.000 }
gfCNCPoint3[7698] = {X 293.5551, Y 9.0595, Z -3.8333, A 0.000, B 0.000, C 0.000 }
gfCNCPoint3[7699] = {X 294.1885, Y 9.6929, Z -3.8333, A 0.000, B 0.000, C 0.000 }
gfCNCPoint3[7700] = {X 294.6650, Y 10.4513, Z -3.8333, A 0.000, B 0.000, C 0.000 }
gfCNCPoint3[7701] = {X 294.9608, Y 11.2967, Z -3.8333, A 0.000, B 0.000, C 0.000 }
gfCNCPoint3[7702] = {X 295.0611, Y 12.1868, Z -3.8333, A 0.000, B 0.000, C 0.000 }
gfCNCPoint3[7703] = {X 295.0609, Y 13.0192, Z -3.8333, A 0.000, B 0.000, C 0.000 }
gfCNCPoint3[7704] = {X 294.9624, Y 13.8611, Z -3.8333, A 0.000, B 0.000, C 0.000 }
gfCNCPoint3[7705] = {X 294.6887, Y 14.6634, Z -3.8333, A 0.000, B 0.000, C 0.000 }
gfCNCPoint3[7706] = {X 294.2521, Y 15.3900, Z -3.8333, A 0.000, B 0.000, C 0.000 }
gfCNCPoint3[7707] = {X 293.6722, Y 16.0083, Z -3.8333, A 0.000, B 0.000, C 0.000 }
gfCNCPoint3[7708] = {X 293.5957, Y 16.0725, Z -3.8333, A 0.000, B 0.000, C 0.000 }
gfCNCPoint3[7709] = {X 293.5177, Y 16.1348, Z -3.8333, A 0.000, B 0.000, C 0.000 }
gfCNCPoint3[7710] = {X 293.5333, Y 16.1922, Z -3.8333, A 0.000, B 0.000, C 0.000 }
gfCNCPoint3[7711] = {X 293.5345, Y 22.5169, Z -3.8333, A 0.000, B 0.000, C 0.000 }
gfCNCPoint3[7712] = {X 293.7676, Y 22.5165, Z -3.8333, A 0.000, B 0.000, C 0.000 }
gfCNCPoint3[7713] = {X 303.0792, Y 22.5173, Z -3.8333, A 0.000, B 0.000, C 0.000 }
gfCNCPoint3[7714] = {X 303.0797, Y 16.1923, Z -3.8333, A 0.000, B 0.000, C 0.000 }
gfCNCPoint3[7715] = {X 303.0955, Y 16.1346, Z -3.8333, A 0.000, B 0.000, C 0.000 }
gfCNCPoint3[7716] = {X 303.0174, Y 16.0723, Z -3.8333, A 0.000, B 0.000, C 0.000 }
gfCNCPoint3[7717] = {X 302.9408, Y 16.0080, Z -3.8333, A 0.000, B 0.000, C 0.000 }
gfCNCPoint3[7718] = {X 302.3549, Y 15.3815, Z -3.8333, A 0.000, B 0.000, C 0.000 }
gfCNCPoint3[7719] = {X 301.9159, Y 14.6445, Z -3.8333, A 0.000, B 0.000, C 0.000 }
gfCNCPoint3[7720] = {X 301.6442, Y 13.8308, Z -3.8333, A 0.000, B 0.000, C 0.000 }
gfCNCPoint3[7721] = {X 301.5523, Y 12.9779, Z -3.8333, A 0.000, B 0.000, C 0.000 }
gfCNCPoint3[7722] = {X 301.5523, Y 12.1868, Z -3.8333, A 0.000, B 0.000, C 0.000 }
gfCNCPoint3[7723] = {X 301.6525, Y 11.2967, Z -3.8333, A 0.000, B 0.000, C 0.000 }
gfCNCPoint3[7724] = {X 301.9484, Y 10.4513, Z -3.8333, A 0.000, B 0.000, C 0.000 }
gfCNCPoint3[7725] = {X 302.4249, Y 9.6929, Z -3.8333, A 0.000, B 0.000, C 0.000 }
gfCNCPoint3[7726] = {X 303.0583, Y 9.0595, Z -3.8333, A 0.000, B 0.000, C 0.000 }
gfCNCPoint3[7727] = {X 303.8167, Y 8.5829, Z -3.8333, A 0.000, B 0.000, C 0.000 }
gfCNCPoint3[7728] = {X 304.6622, Y 8.2871, Z -3.8333, A 0.000, B 0.000, C 0.000 }
gfCNCPoint3[7729] = {X 305.5523, Y 8.1868, Z -3.8333, A 0.000, B 0.000, C 0.000 }
gfCNCPoint3[7730] = {X 311.9957, Y 8.1868, Z -3.8333, A 0.000, B 0.000, C 0.000 }
gfCNCPoint3[7731] = {X 312.8858, Y 8.2871, Z -3.8333, A 0.000, B 0.000, C 0.000 }
gfCNCPoint3[7732] = {X 313.7313, Y 8.5829, Z -3.8333, A 0.000, B 0.000, C 0.000 }
gfCNCPoint3[7733] = {X 314.4897, Y 9.0595, Z -3.8333, A 0.000, B 0.000, C 0.000 }
gfCNCPoint3[7734] = {X 315.1230, Y 9.6929, Z -3.8333, A 0.000, B 0.000, C 0.000 }
gfCNCPoint3[7735] = {X 315.5996, Y 10.4513, Z -3.8333, A 0.000, B 0.000, C 0.000 }
gfCNCPoint3[7736] = {X 315.8954, Y 11.2967, Z -3.8333, A 0.000, B 0.000, C 0.000 }
gfCNCPoint3[7737] = {X 315.9957, Y 12.1868, Z -3.8333, A 0.000, B 0.000, C 0.000 }
gfCNCPoint3[7738] = {X 315.9955, Y 13.0192, Z -3.8333, A 0.000, B 0.000, C 0.000 }
gfCNCPoint3[7739] = {X 315.8970, Y 13.8611, Z -3.8333, A 0.000, B 0.000, C 0.000 }
gfCNCPoint3[7740] = {X 315.6234, Y 14.6633, Z -3.8333, A 0.000, B 0.000, C 0.000 }
gfCNCPoint3[7741] = {X 315.1868, Y 15.3899, Z -3.8333, A 0.000, B 0.000, C 0.000 }
gfCNCPoint3[7742] = {X 314.6069, Y 16.0081, Z -3.8333, A 0.000, B 0.000, C 0.000 }
gfCNCPoint3[7743] = {X 314.5389, Y 16.0655, Z -3.8333, A 0.000, B 0.000, C 0.000 }
gfCNCPoint3[7744] = {X 314.4695, Y 16.1213, Z -3.8333, A 0.000, B 0.000, C 0.000 }
gfCNCPoint3[7745] = {X 314.4680, Y 16.3112, Z -3.8333, A 0.000, B 0.000, C 0.000 }
gfCNCPoint3[7746] = {X 314.4678, Y 41.0666, Z -3.8333, A 0.000, B 0.000, C 0.000 }
gfCNCPoint3[7747] = {X 314.6067, Y 41.1785, Z -3.8333, A 0.000, B 0.000, C 0.000 }
gfCNCPoint3[7748] = {X 315.1929, Y 41.8050, Z -3.8333, A 0.000, B 0.000, C 0.000 }
gfCNCPoint3[7749] = {X 315.6319, Y 42.5421, Z -3.8333, A 0.000, B 0.000, C 0.000 }
gfCNCPoint3[7750] = {X 315.9037, Y 43.3559, Z -3.8333, A 0.000, B 0.000, C 0.000 }
gfCNCPoint3[7751] = {X 315.9957, Y 44.2089, Z -3.8333, A 0.000, B 0.000, C 0.000 }
gfCNCPoint3[7752] = {X 315.9957, Y 45.0000, Z -3.8333, A 0.000, B 0.000, C 0.000 }
gfCNCPoint3[7753] = {X 315.8954, Y 45.8901, Z -3.8333, A 0.000, B 0.000, C 0.000 }
gfCNCPoint3[7754] = {X 315.5996, Y 46.7355, Z -3.8333, A 0.000, B 0.000, C 0.000 }
gfCNCPoint3[7755] = {X 315.1230, Y 47.4940, Z -3.8333, A 0.000, B 0.000, C 0.000 }
gfCNCPoint3[7756] = {X 314.4897, Y 48.1273, Z -3.8333, A 0.000, B 0.000, C 0.000 }
gfCNCPoint3[7757] = {X 313.7313, Y 48.6039, Z -3.8333, A 0.000, B 0.000, C 0.000 }
gfCNCPoint3[7758] = {X 312.8858, Y 48.8997, Z -3.8333, A 0.000, B 0.000, C 0.000 }
gfCNCPoint3[7759] = {X 311.9957, Y 49.0000, Z -3.8333, A 0.000, B 0.000, C 0.000 }
gfCNCPoint3[7760] = {X 305.5523, Y 49.0000, Z -3.8333, A 0.000, B 0.000, C 0.000 }
gfCNCPoint3[7761] = {X 304.6622, Y 48.8997, Z -3.8333, A 0.000, B 0.000, C 0.000 }
gfCNCPoint3[7762] = {X 303.8167, Y 48.6039, Z -3.8333, A 0.000, B 0.000, C 0.000 }
gfCNCPoint3[7763] = {X 303.0583, Y 48.1273, Z -3.8333, A 0.000, B 0.000, C 0.000 }
gfCNCPoint3[7764] = {X 302.4249, Y 47.4939, Z -3.8333, A 0.000, B 0.000, C 0.000 }
gfCNCPoint3[7765] = {X 301.9484, Y 46.7355, Z -3.8333, A 0.000, B 0.000, C 0.000 }
gfCNCPoint3[7766] = {X 301.6525, Y 45.8900, Z -3.8333, A 0.000, B 0.000, C 0.000 }
gfCNCPoint3[7767] = {X 301.5523, Y 45.0000, Z -3.8333, A 0.000, B 0.000, C 0.000 }
gfCNCPoint3[7768] = {X 301.5523, Y 44.2089, Z -3.8333, A 0.000, B 0.000, C 0.000 }
gfCNCPoint3[7769] = {X 301.6699, Y 43.3029, Z -3.8333, A 0.000, B 0.000, C 0.000 }
gfCNCPoint3[7770] = {X 301.9739, Y 42.4415, Z -3.8333, A 0.000, B 0.000, C 0.000 }
gfCNCPoint3[7771] = {X 302.4510, Y 41.6623, Z -3.8333, A 0.000, B 0.000, C 0.000 }
gfCNCPoint3[7772] = {X 303.0801, Y 40.9999, Z -3.8333, A 0.000, B 0.000, C 0.000 }
gfCNCPoint3[7773] = {X 303.0801, Y 33.7143, Z -3.8333, A 0.000, B 0.000, C 0.000 }
gfCNCPoint3[7774] = {X 293.9342, Y 33.7143, Z -3.8333, A 0.000, B 0.000, C 0.000 }
gfCNCPoint3[7775] = {X 293.5343, Y 33.7136, Z -3.8333, A 0.000, B 0.000, C 0.000 }
gfCNCPoint3[7776] = {X 293.5333, Y 41.0521, Z -3.8333, A 0.000, B 0.000, C 0.000 }
gfCNCPoint3[7777] = {X 294.1706, Y 41.6934, Z -3.8333, A 0.000, B 0.000, C 0.000 }
gfCNCPoint3[7778] = {X 294.6519, Y 42.4589, Z -3.8333, A 0.000, B 0.000, C 0.000 }
gfCNCPoint3[7779] = {X 294.9536, Y 43.3112, Z -3.8333, A 0.000, B 0.000, C 0.000 }
gfCNCPoint3[7780] = {X 295.0611, Y 44.2089, Z -3.8333, A 0.000, B 0.000, C 0.000 }
gfCNCPoint3[7781] = {X 295.0611, Y 45.0000, Z -3.8333, A 0.000, B 0.000, C 0.000 }
gfCNCPoint3[7782] = {X 294.9608, Y 45.8901, Z -3.8333, A 0.000, B 0.000, C 0.000 }
gfCNCPoint3[7783] = {X 294.6650, Y 46.7355, Z -3.8333, A 0.000, B 0.000, C 0.000 }
gfCNCPoint3[7784] = {X 294.1885, Y 47.4940, Z -3.8333, A 0.000, B 0.000, C 0.000 }
gfCNCPoint3[7785] = {X 293.5551, Y 48.1273, Z -3.8333, A 0.000, B 0.000, C 0.000 }
gfCNCPoint3[7786] = {X 292.7967, Y 48.6039, Z -3.8333, A 0.000, B 0.000, C 0.000 }
gfCNCPoint3[7787] = {X 291.9512, Y 48.8997, Z -3.8333, A 0.000, B 0.000, C 0.000 }
gfCNCPoint3[7788] = {X 291.0611, Y 49.0000, Z -3.8333, A 0.000, B 0.000, C 0.000 }
gfCNCPoint3[7789] = {X 284.6177, Y 49.0000, Z -3.8333, A 0.000, B 0.000, C 0.000 }
gfCNCPoint3[7790] = {X 283.7276, Y 48.8997, Z -3.8333, A 0.000, B 0.000, C 0.000 }
gfCNCPoint3[7791] = {X 282.8821, Y 48.6039, Z -3.8333, A 0.000, B 0.000, C 0.000 }
gfCNCPoint3[7792] = {X 282.1237, Y 48.1273, Z -3.8333, A 0.000, B 0.000, C 0.000 }
gfCNCPoint3[7793] = {X 281.4903, Y 47.4939, Z -3.8333, A 0.000, B 0.000, C 0.000 }
gfCNCPoint3[7794] = {X 281.0138, Y 46.7355, Z -3.8333, A 0.000, B 0.000, C 0.000 }
gfCNCPoint3[7795] = {X 280.7180, Y 45.8901, Z -3.8333, A 0.000, B 0.000, C 0.000 }
gfCNCPoint3[7796] = {X 280.6177, Y 45.0000, Z -3.8333, A 0.000, B 0.000, C 0.000 }
gfCNCPoint3[7797] = {X 280.6177, Y 44.2089, Z -3.8333, A 0.000, B 0.000, C 0.000 }
gfCNCPoint3[7798] = {X 280.7231, Y 43.3126, Z -3.8333, A 0.000, B 0.000, C 0.000 }
gfCNCPoint3[7799] = {X 281.0243, Y 42.4618, Z -3.8333, A 0.000, B 0.000, C 0.000 }
gfCNCPoint3[7800] = {X 281.5065, Y 41.6989, Z -3.8333, A 0.000, B 0.000, C 0.000 }
gfCNCPoint3[7801] = {X 282.1456, Y 41.0618, Z -3.8333, A 0.000, B 0.000, C 0.000 }
gfCNCPoint3[7802] = {X 282.1454, Y 28.5926, Z -3.8333, A 0.000, B 0.000, C 0.000 }
gfCNCPoint3[7803] = {X 278.0654, Y 28.5927, Z -3.8333, A 0.000, B 0.000, C 0.000 }
gfCNCPoint3[7804] = {X 278.0654, Y 28.5927, Z -0.8333, A 0.000, B 0.000, C 0.000 }
gfCNCPoint3[7805] = {X 278.0654, Y 28.5927, Z 11.0000, A 0.000, B 0.000, C 0.000 }
gfCNCPoint3[7806] = {X 353.3542, Y 107.0433, Z 11.0000, A 0.000, B 0.000, C 0.000 }
gfCNCPoint3[7807] = {X 353.3542, Y 107.0433, Z -0.8333, A 0.000, B 0.000, C 0.000 }
gfCNCPoint3[7808] = {X 353.3542, Y 107.0433, Z -3.8333, A 0.000, B 0.000, C 0.000 }
gfCNCPoint3[7809] = {X 353.2425, Y 102.9649, Z -3.8333, A 0.000, B 0.000, C 0.000 }
gfCNCPoint3[7810] = {X 347.7202, Y 103.0334, Z -3.8333, A 0.000, B 0.000, C 0.000 }
gfCNCPoint3[7811] = {X 342.1983, Y 102.9367, Z -3.8333, A 0.000, B 0.000, C 0.000 }
gfCNCPoint3[7812] = {X 336.6818, Y 102.6748, Z -3.8333, A 0.000, B 0.000, C 0.000 }
gfCNCPoint3[7813] = {X 333.1921, Y 102.3986, Z -3.8333, A 0.000, B 0.000, C 0.000 }
gfCNCPoint3[7814] = {X 329.7160, Y 101.9856, Z -3.8333, A 0.000, B 0.000, C 0.000 }
gfCNCPoint3[7815] = {X 326.2587, Y 101.4366, Z -3.8333, A 0.000, B 0.000, C 0.000 }
gfCNCPoint3[7816] = {X 323.4089, Y 100.8329, Z -3.8333, A 0.000, B 0.000, C 0.000 }
gfCNCPoint3[7817] = {X 320.6115, Y 100.0199, Z -3.8333, A 0.000, B 0.000, C 0.000 }
gfCNCPoint3[7818] = {X 317.8819, Y 99.0022, Z -3.8333, A 0.000, B 0.000, C 0.000 }
gfCNCPoint3[7819] = {X 316.3695, Y 98.3037, Z -3.8333, A 0.000, B 0.000, C 0.000 }
gfCNCPoint3[7820] = {X 314.9205, Y 97.4817, Z -3.8333, A 0.000, B 0.000, C 0.000 }
gfCNCPoint3[7821] = {X 313.5451, Y 96.5418, Z -3.8333, A 0.000, B 0.000, C 0.000 }
gfCNCPoint3[7822] = {X 312.2526, Y 95.4907, Z -3.8333, A 0.000, B 0.000, C 0.000 }
gfCNCPoint3[7823] = {X 311.2489, Y 94.4924, Z -3.8333, A 0.000, B 0.000, C 0.000 }
gfCNCPoint3[7824] = {X 310.3707, Y 93.3820, Z -3.8333, A 0.000, B 0.000, C 0.000 }
gfCNCPoint3[7825] = {X 309.6303, Y 92.1753, Z -3.8333, A 0.000, B 0.000, C 0.000 }
gfCNCPoint3[7826] = {X 309.0383, Y 90.8894, Z -3.8333, A 0.000, B 0.000, C 0.000 }
gfCNCPoint3[7827] = {X 308.6030, Y 89.5423, Z -3.8333, A 0.000, B 0.000, C 0.000 }
gfCNCPoint3[7828] = {X 308.2595, Y 87.9192, Z -3.8333, A 0.000, B 0.000, C 0.000 }
gfCNCPoint3[7829] = {X 308.0566, Y 86.2727, Z -3.8333, A 0.000, B 0.000, C 0.000 }
gfCNCPoint3[7830] = {X 307.9957, Y 84.6148, Z -3.8333, A 0.000, B 0.000, C 0.000 }
gfCNCPoint3[7831] = {X 307.9970, Y 63.2123, Z -3.8333, A 0.000, B 0.000, C 0.000 }
gfCNCPoint3[7832] = {X 307.1454, Y 63.0032, Z -3.8333, A 0.000, B 0.000, C 0.000 }
gfCNCPoint3[7833] = {X 306.3536, Y 62.6264, Z -3.8333, A 0.000, B 0.000, C 0.000 }
gfCNCPoint3[7834] = {X 305.6542, Y 62.0974, Z -3.8333, A 0.000, B 0.000, C 0.000 }
gfCNCPoint3[7835] = {X 305.0760, Y 61.4382, Z -3.8333, A 0.000, B 0.000, C 0.000 }
gfCNCPoint3[7836] = {X 304.6429, Y 60.6757, Z -3.8333, A 0.000, B 0.000, C 0.000 }
gfCNCPoint3[7837] = {X 304.3726, Y 59.8415, Z -3.8333, A 0.000, B 0.000, C 0.000 }
gfCNCPoint3[7838] = {X 304.2764, Y 58.9699, Z -3.8333, A 0.000, B 0.000, C 0.000 }
gfCNCPoint3[7839] = {X 304.2762, Y 58.0000, Z -3.8333, A 0.000, B 0.000, C 0.000 }
gfCNCPoint3[7840] = {X 304.3845, Y 57.0387, Z -3.8333, A 0.000, B 0.000, C 0.000 }
gfCNCPoint3[7841] = {X 304.7040, Y 56.1256, Z -3.8333, A 0.000, B 0.000, C 0.000 }
gfCNCPoint3[7842] = {X 305.2187, Y 55.3065, Z -3.8333, A 0.000, B 0.000, C 0.000 }
gfCNCPoint3[7843] = {X 305.9027, Y 54.6225, Z -3.8333, A 0.000, B 0.000, C 0.000 }
gfCNCPoint3[7844] = {X 306.7218, Y 54.1078, Z -3.8333, A 0.000, B 0.000, C 0.000 }
gfCNCPoint3[7845] = {X 307.6349, Y 53.7883, Z -3.8333, A 0.000, B 0.000, C 0.000 }
gfCNCPoint3[7846] = {X 308.5962, Y 53.6800, Z -3.8333, A 0.000, B 0.000, C 0.000 }
gfCNCPoint3[7847] = {X 324.3107, Y 53.6800, Z -3.8333, A 0.000, B 0.000, C 0.000 }
gfCNCPoint3[7848] = {X 325.2720, Y 53.7883, Z -3.8333, A 0.000, B 0.000, C 0.000 }
gfCNCPoint3[7849] = {X 326.1851, Y 54.1078, Z -3.8333, A 0.000, B 0.000, C 0.000 }
gfCNCPoint3[7850] = {X 327.0042, Y 54.6225, Z -3.8333, A 0.000, B 0.000, C 0.000 }
gfCNCPoint3[7851] = {X 327.6882, Y 55.3065, Z -3.8333, A 0.000, B 0.000, C 0.000 }
gfCNCPoint3[7852] = {X 328.2029, Y 56.1256, Z -3.8333, A 0.000, B 0.000, C 0.000 }
gfCNCPoint3[7853] = {X 328.5224, Y 57.0387, Z -3.8333, A 0.000, B 0.000, C 0.000 }
gfCNCPoint3[7854] = {X 328.6307, Y 58.0000, Z -3.8333, A 0.000, B 0.000, C 0.000 }
gfCNCPoint3[7855] = {X 328.6307, Y 58.9360, Z -3.8333, A 0.000, B 0.000, C 0.000 }
gfCNCPoint3[7856] = {X 328.5365, Y 59.8122, Z -3.8333, A 0.000, B 0.000, C 0.000 }
gfCNCPoint3[7857] = {X 328.2679, Y 60.6516, Z -3.8333, A 0.000, B 0.000, C 0.000 }
gfCNCPoint3[7858] = {X 327.8360, Y 61.4198, Z -3.8333, A 0.000, B 0.000, C 0.000 }
gfCNCPoint3[7859] = {X 327.2584, Y 62.0854, Z -3.8333, A 0.000, B 0.000, C 0.000 }
gfCNCPoint3[7860] = {X 326.5587, Y 62.6212, Z -3.8333, A 0.000, B 0.000, C 0.000 }
gfCNCPoint3[7861] = {X 325.7655, Y 63.0054, Z -3.8333, A 0.000, B 0.000, C 0.000 }
gfCNCPoint3[7862] = {X 324.9113, Y 63.2221, Z -3.8333, A 0.000, B 0.000, C 0.000 }
gfCNCPoint3[7863] = {X 324.9129, Y 83.2296, Z -3.8333, A 0.000, B 0.000, C 0.000 }
gfCNCPoint3[7864] = {X 324.9264, Y 84.6148, Z -3.8333, A 0.000, B 0.000, C 0.000 }
gfCNCPoint3[7865] = {X 325.0038, Y 85.8500, Z -3.8333, A 0.000, B 0.000, C 0.000 }
gfCNCPoint3[7866] = {X 325.2261, Y 87.0675, Z -3.8333, A 0.000, B 0.000, C 0.000 }
gfCNCPoint3[7867] = {X 325.4715, Y 87.3363, Z -3.8333, A 0.000, B 0.000, C 0.000 }
gfCNCPoint3[7868] = {X 325.7737, Y 87.5392, Z -3.8333, A 0.000, B 0.000, C 0.000 }
gfCNCPoint3[7869] = {X 326.2242, Y 87.7937, Z -3.8333, A 0.000, B 0.000, C 0.000 }
gfCNCPoint3[7870] = {X 327.6622, Y 88.3905, Z -3.8333, A 0.000, B 0.000, C 0.000 }
gfCNCPoint3[7871] = {X 329.1569, Y 88.8264, Z -3.8333, A 0.000, B 0.000, C 0.000 }
gfCNCPoint3[7872] = {X 332.2329, Y 89.4422, Z -3.8333, A 0.000, B 0.000, C 0.000 }
gfCNCPoint3[7873] = {X 335.3453, Y 89.8350, Z -3.8333, A 0.000, B 0.000, C 0.000 }
gfCNCPoint3[7874] = {X 339.4834, Y 90.1553, Z -3.8333, A 0.000, B 0.000, C 0.000 }
gfCNCPoint3[7875] = {X 343.6300, Y 90.3349, Z -3.8333, A 0.000, B 0.000, C 0.000 }
gfCNCPoint3[7876] = {X 347.7803, Y 90.3737, Z -3.8333, A 0.000, B 0.000, C 0.000 }
gfCNCPoint3[7877] = {X 352.1620, Y 90.3353, Z -3.8333, A 0.000, B 0.000, C 0.000 }
gfCNCPoint3[7878] = {X 356.5395, Y 90.1394, Z -3.8333, A 0.000, B 0.000, C 0.000 }
gfCNCPoint3[7879] = {X 360.9071, Y 89.7864, Z -3.8333, A 0.000, B 0.000, C 0.000 }
gfCNCPoint3[7880] = {X 363.2212, Y 89.4986, Z -3.8333, A 0.000, B 0.000, C 0.000 }
gfCNCPoint3[7881] = {X 365.5139, Y 89.0722, Z -3.8333, A 0.000, B 0.000, C 0.000 }
gfCNCPoint3[7882] = {X 367.7768, Y 88.5088, Z -3.8333, A 0.000, B 0.000, C 0.000 }
gfCNCPoint3[7883] = {X 368.7088, Y 88.1955, Z -3.8333, A 0.000, B 0.000, C 0.000 }
gfCNCPoint3[7884] = {X 369.5998, Y 87.7797, Z -3.8333, A 0.000, B 0.000, C 0.000 }
gfCNCPoint3[7885] = {X 370.4385, Y 87.2665, Z -3.8333, A 0.000, B 0.000, C 0.000 }
gfCNCPoint3[7886] = {X 370.5883, Y 87.1106, Z -3.8333, A 0.000, B 0.000, C 0.000 }
gfCNCPoint3[7887] = {X 370.6656, Y 86.9086, Z -3.8333, A 0.000, B 0.000, C 0.000 }
gfCNCPoint3[7888] = {X 370.8567, Y 85.3736, Z -3.8333, A 0.000, B 0.000, C 0.000 }
gfCNCPoint3[7889] = {X 370.9204, Y 83.8281, Z -3.8333, A 0.000, B 0.000, C 0.000 }
gfCNCPoint3[7890] = {X 370.9206, Y 63.2124, Z -3.8333, A 0.000, B 0.000, C 0.000 }
gfCNCPoint3[7891] = {X 370.0689, Y 63.0033, Z -3.8333, A 0.000, B 0.000, C 0.000 }
gfCNCPoint3[7892] = {X 369.2770, Y 62.6266, Z -3.8333, A 0.000, B 0.000, C 0.000 }
gfCNCPoint3[7893] = {X 368.5774, Y 62.0976, Z -3.8333, A 0.000, B 0.000, C 0.000 }
gfCNCPoint3[7894] = {X 367.9992, Y 61.4383, Z -3.8333, A 0.000, B 0.000, C 0.000 }
gfCNCPoint3[7895] = {X 367.5659, Y 60.6758, Z -3.8333, A 0.000, B 0.000, C 0.000 }
gfCNCPoint3[7896] = {X 367.2957, Y 59.8414, Z -3.8333, A 0.000, B 0.000, C 0.000 }
gfCNCPoint3[7897] = {X 367.1994, Y 58.9697, Z -3.8333, A 0.000, B 0.000, C 0.000 }
gfCNCPoint3[7898] = {X 367.1993, Y 58.0000, Z -3.8333, A 0.000, B 0.000, C 0.000 }
gfCNCPoint3[7899] = {X 367.3076, Y 57.0387, Z -3.8333, A 0.000, B 0.000, C 0.000 }
gfCNCPoint3[7900] = {X 367.6271, Y 56.1256, Z -3.8333, A 0.000, B 0.000, C 0.000 }
gfCNCPoint3[7901] = {X 368.1418, Y 55.3065, Z -3.8333, A 0.000, B 0.000, C 0.000 }
gfCNCPoint3[7902] = {X 368.8258, Y 54.6225, Z -3.8333, A 0.000, B 0.000, C 0.000 }
gfCNCPoint3[7903] = {X 369.6449, Y 54.1078, Z -3.8333, A 0.000, B 0.000, C 0.000 }
gfCNCPoint3[7904] = {X 370.5580, Y 53.7883, Z -3.8333, A 0.000, B 0.000, C 0.000 }
gfCNCPoint3[7905] = {X 371.5193, Y 53.6800, Z -3.8333, A 0.000, B 0.000, C 0.000 }
gfCNCPoint3[7906] = {X 388.0597, Y 53.6800, Z -3.8333, A 0.000, B 0.000, C 0.000 }
gfCNCPoint3[7907] = {X 389.0210, Y 53.7883, Z -3.8333, A 0.000, B 0.000, C 0.000 }
gfCNCPoint3[7908] = {X 389.9341, Y 54.1078, Z -3.8333, A 0.000, B 0.000, C 0.000 }
gfCNCPoint3[7909] = {X 390.7532, Y 54.6225, Z -3.8333, A 0.000, B 0.000, C 0.000 }
gfCNCPoint3[7910] = {X 391.4372, Y 55.3065, Z -3.8333, A 0.000, B 0.000, C 0.000 }
gfCNCPoint3[7911] = {X 391.9519, Y 56.1256, Z -3.8333, A 0.000, B 0.000, C 0.000 }
gfCNCPoint3[7912] = {X 392.2714, Y 57.0387, Z -3.8333, A 0.000, B 0.000, C 0.000 }
gfCNCPoint3[7913] = {X 392.3797, Y 58.0000, Z -3.8333, A 0.000, B 0.000, C 0.000 }
gfCNCPoint3[7914] = {X 392.3797, Y 58.9342, Z -3.8333, A 0.000, B 0.000, C 0.000 }
gfCNCPoint3[7915] = {X 392.2652, Y 59.9219, Z -3.8333, A 0.000, B 0.000, C 0.000 }
gfCNCPoint3[7916] = {X 391.9280, Y 60.8573, Z -3.8333, A 0.000, B 0.000, C 0.000 }
gfCNCPoint3[7917] = {X 391.4847, Y 61.5690, Z -3.8333, A 0.000, B 0.000, C 0.000 }
gfCNCPoint3[7918] = {X 390.9129, Y 62.1823, Z -3.8333, A 0.000, B 0.000, C 0.000 }
gfCNCPoint3[7919] = {X 390.2339, Y 62.6742, Z -3.8333, A 0.000, B 0.000, C 0.000 }
gfCNCPoint3[7920] = {X 389.4730, Y 63.0265, Z -3.8333, A 0.000, B 0.000, C 0.000 }
gfCNCPoint3[7921] = {X 388.6586, Y 63.2259, Z -3.8333, A 0.000, B 0.000, C 0.000 }
gfCNCPoint3[7922] = {X 388.6566, Y 84.6148, Z -3.8333, A 0.000, B 0.000, C 0.000 }
gfCNCPoint3[7923] = {X 388.5967, Y 86.2731, Z -3.8333, A 0.000, B 0.000, C 0.000 }
gfCNCPoint3[7924] = {X 388.3923, Y 87.9200, Z -3.8333, A 0.000, B 0.000, C 0.000 }
gfCNCPoint3[7925] = {X 388.0451, Y 89.5427, Z -3.8333, A 0.000, B 0.000, C 0.000 }
gfCNCPoint3[7926] = {X 387.5130, Y 91.1300, Z -3.8333, A 0.000, B 0.000, C 0.000 }
gfCNCPoint3[7927] = {X 386.7634, Y 92.6269, Z -3.8333, A 0.000, B 0.000, C 0.000 }
gfCNCPoint3[7928] = {X 385.8113, Y 94.0039, Z -3.8333, A 0.000, B 0.000, C 0.000 }
gfCNCPoint3[7929] = {X 384.6755, Y 95.2338, Z -3.8333, A 0.000, B 0.000, C 0.000 }
gfCNCPoint3[7930] = {X 383.1611, Y 96.5097, Z -3.8333, A 0.000, B 0.000, C 0.000 }
gfCNCPoint3[7931] = {X 381.5199, Y 97.6177, Z -3.8333, A 0.000, B 0.000, C 0.000 }
gfCNCPoint3[7932] = {X 379.7703, Y 98.5452, Z -3.8333, A 0.000, B 0.000, C 0.000 }
gfCNCPoint3[7933] = {X 377.4992, Y 99.5014, Z -3.8333, A 0.000, B 0.000, C 0.000 }
gfCNCPoint3[7934] = {X 375.1651, Y 100.2916, Z -3.8333, A 0.000, B 0.000, C 0.000 }
gfCNCPoint3[7935] = {X 372.7802, Y 100.9120, Z -3.8333, A 0.000, B 0.000, C 0.000 }
gfCNCPoint3[7936] = {X 368.9685, Y 101.6494, Z -3.8333, A 0.000, B 0.000, C 0.000 }
gfCNCPoint3[7937] = {X 365.1257, Y 102.2027, Z -3.8333, A 0.000, B 0.000, C 0.000 }
gfCNCPoint3[7938] = {X 361.2608, Y 102.5707, Z -3.8333, A 0.000, B 0.000, C 0.000 }
gfCNCPoint3[7939] = {X 357.2538, Y 102.8114, Z -3.8333, A 0.000, B 0.000, C 0.000 }
gfCNCPoint3[7940] = {X 353.2425, Y 102.9649, Z -3.8333, A 0.000, B 0.000, C 0.000 }
gfCNCPoint3[7941] = {X 353.3520, Y 106.9634, Z -3.8333, A 0.000, B 0.000, C 0.000 }
gfCNCPoint3[7942] = {X 353.2403, Y 102.8849, Z -3.8333, A 0.000, B 0.000, C 0.000 }
gfCNCPoint3[7943] = {X 347.7204, Y 102.9534, Z -3.8333, A 0.000, B 0.000, C 0.000 }
gfCNCPoint3[7944] = {X 342.2009, Y 102.8567, Z -3.8333, A 0.000, B 0.000, C 0.000 }
gfCNCPoint3[7945] = {X 336.6868, Y 102.5949, Z -3.8333, A 0.000, B 0.000, C 0.000 }
gfCNCPoint3[7946] = {X 333.2001, Y 102.3189, Z -3.8333, A 0.000, B 0.000, C 0.000 }
gfCNCPoint3[7947] = {X 329.7269, Y 101.9064, Z -3.8333, A 0.000, B 0.000, C 0.000 }
gfCNCPoint3[7948] = {X 326.2726, Y 101.3578, Z -3.8333, A 0.000, B 0.000, C 0.000 }
gfCNCPoint3[7949] = {X 323.4285, Y 100.7553, Z -3.8333, A 0.000, B 0.000, C 0.000 }
gfCNCPoint3[7950] = {X 320.6367, Y 99.9440, Z -3.8333, A 0.000, B 0.000, C 0.000 }
gfCNCPoint3[7951] = {X 317.9126, Y 98.9283, Z -3.8333, A 0.000, B 0.000, C 0.000 }
gfCNCPoint3[7952] = {X 316.4062, Y 98.2326, Z -3.8333, A 0.000, B 0.000, C 0.000 }
gfCNCPoint3[7953] = {X 314.9630, Y 97.4139, Z -3.8333, A 0.000, B 0.000, C 0.000 }
gfCNCPoint3[7954] = {X 313.5929, Y 96.4778, Z -3.8333, A 0.000, B 0.000, C 0.000 }
gfCNCPoint3[7955] = {X 312.3057, Y 95.4308, Z -3.8333, A 0.000, B 0.000, C 0.000 }
gfCNCPoint3[7956] = {X 311.3086, Y 94.4391, Z -3.8333, A 0.000, B 0.000, C 0.000 }
gfCNCPoint3[7957] = {X 310.4363, Y 93.3362, Z -3.8333, A 0.000, B 0.000, C 0.000 }
gfCNCPoint3[7958] = {X 309.7009, Y 92.1376, Z -3.8333, A 0.000, B 0.000, C 0.000 }
gfCNCPoint3[7959] = {X 309.1128, Y 90.8603, Z -3.8333, A 0.000, B 0.000, C 0.000 }
gfCNCPoint3[7960] = {X 308.6804, Y 89.5222, Z -3.8333, A 0.000, B 0.000, C 0.000 }
gfCNCPoint3[7961] = {X 308.3384, Y 87.9059, Z -3.8333, A 0.000, B 0.000, C 0.000 }
gfCNCPoint3[7962] = {X 308.1363, Y 86.2661, Z -3.8333, A 0.000, B 0.000, C 0.000 }
gfCNCPoint3[7963] = {X 308.0757, Y 84.6151, Z -3.8333, A 0.000, B 0.000, C 0.000 }
gfCNCPoint3[7964] = {X 308.0770, Y 63.1421, Z -3.8333, A 0.000, B 0.000, C 0.000 }
gfCNCPoint3[7965] = {X 307.2285, Y 62.9474, Z -3.8333, A 0.000, B 0.000, C 0.000 }
gfCNCPoint3[7966] = {X 306.4377, Y 62.5835, Z -3.8333, A 0.000, B 0.000, C 0.000 }
gfCNCPoint3[7967] = {X 305.7379, Y 62.0658, Z -3.8333, A 0.000, B 0.000, C 0.000 }
gfCNCPoint3[7968] = {X 305.1586, Y 61.4160, Z -3.8333, A 0.000, B 0.000, C 0.000 }
gfCNCPoint3[7969] = {X 304.7241, Y 60.6616, Z -3.8333, A 0.000, B 0.000, C 0.000 }
gfCNCPoint3[7970] = {X 304.4529, Y 59.8344, Z -3.8333, A 0.000, B 0.000, C 0.000 }
gfCNCPoint3[7971] = {X 304.3564, Y 58.9693, Z -3.8333, A 0.000, B 0.000, C 0.000 }
gfCNCPoint3[7972] = {X 304.3562, Y 58.0000, Z -3.8333, A 0.000, B 0.000, C 0.000 }
gfCNCPoint3[7973] = {X 304.4625, Y 57.0565, Z -3.8333, A 0.000, B 0.000, C 0.000 }
gfCNCPoint3[7974] = {X 304.7761, Y 56.1603, Z -3.8333, A 0.000, B 0.000, C 0.000 }
gfCNCPoint3[7975] = {X 305.2813, Y 55.3564, Z -3.8333, A 0.000, B 0.000, C 0.000 }
gfCNCPoint3[7976] = {X 305.9526, Y 54.6850, Z -3.8333, A 0.000, B 0.000, C 0.000 }
gfCNCPoint3[7977] = {X 306.7566, Y 54.1799, Z -3.8333, A 0.000, B 0.000, C 0.000 }
gfCNCPoint3[7978] = {X 307.6527, Y 53.8663, Z -3.8333, A 0.000, B 0.000, C 0.000 }
gfCNCPoint3[7979] = {X 308.5962, Y 53.7600, Z -3.8333, A 0.000, B 0.000, C 0.000 }
gfCNCPoint3[7980] = {X 324.3107, Y 53.7600, Z -3.8333, A 0.000, B 0.000, C 0.000 }
gfCNCPoint3[7981] = {X 325.2542, Y 53.8663, Z -3.8333, A 0.000, B 0.000, C 0.000 }
gfCNCPoint3[7982] = {X 326.1504, Y 54.1799, Z -3.8333, A 0.000, B 0.000, C 0.000 }
gfCNCPoint3[7983] = {X 326.9543, Y 54.6850, Z -3.8333, A 0.000, B 0.000, C 0.000 }
gfCNCPoint3[7984] = {X 327.6257, Y 55.3564, Z -3.8333, A 0.000, B 0.000, C 0.000 }
gfCNCPoint3[7985] = {X 328.1308, Y 56.1603, Z -3.8333, A 0.000, B 0.000, C 0.000 }
gfCNCPoint3[7986] = {X 328.4444, Y 57.0565, Z -3.8333, A 0.000, B 0.000, C 0.000 }
gfCNCPoint3[7987] = {X 328.5507, Y 58.0000, Z -3.8333, A 0.000, B 0.000, C 0.000 }
gfCNCPoint3[7988] = {X 328.5507, Y 58.9355, Z -3.8333, A 0.000, B 0.000, C 0.000 }
gfCNCPoint3[7989] = {X 328.4561, Y 59.8053, Z -3.8333, A 0.000, B 0.000, C 0.000 }
gfCNCPoint3[7990] = {X 328.1866, Y 60.6377, Z -3.8333, A 0.000, B 0.000, C 0.000 }
gfCNCPoint3[7991] = {X 327.7535, Y 61.3978, Z -3.8333, A 0.000, B 0.000, C 0.000 }
gfCNCPoint3[7992] = {X 327.1748, Y 62.0540, Z -3.8333, A 0.000, B 0.000, C 0.000 }
gfCNCPoint3[7993] = {X 326.4747, Y 62.5787, Z -3.8333, A 0.000, B 0.000, C 0.000 }
gfCNCPoint3[7994] = {X 325.6825, Y 62.9501, Z -3.8333, A 0.000, B 0.000, C 0.000 }
gfCNCPoint3[7995] = {X 324.8313, Y 63.1525, Z -3.8333, A 0.000, B 0.000, C 0.000 }
gfCNCPoint3[7996] = {X 324.8329, Y 83.2300, Z -3.8333, A 0.000, B 0.000, C 0.000 }
gfCNCPoint3[7997] = {X 324.8464, Y 84.6150, Z -3.8333, A 0.000, B 0.000, C 0.000 }
gfCNCPoint3[7998] = {X 324.9253, Y 85.8672, Z -3.8333, A 0.000, B 0.000, C 0.000 }
gfCNCPoint3[7999] = {X 325.1520, Y 87.1013, Z -3.8333, A 0.000, B 0.000, C 0.000 }
gfCNCPoint3[8000] = {X 325.4128, Y 87.3913, Z -3.8333, A 0.000, B 0.000, C 0.000 }
gfCNCPoint3[8001] = {X 325.7358, Y 87.6097, Z -3.8333, A 0.000, B 0.000, C 0.000 }
gfCNCPoint3[8002] = {X 326.1872, Y 87.8647, Z -3.8333, A 0.000, B 0.000, C 0.000 }
gfCNCPoint3[8003] = {X 327.6344, Y 88.4656, Z -3.8333, A 0.000, B 0.000, C 0.000 }
gfCNCPoint3[8004] = {X 329.1388, Y 88.9043, Z -3.8333, A 0.000, B 0.000, C 0.000 }
gfCNCPoint3[8005] = {X 332.2202, Y 89.5212, Z -3.8333, A 0.000, B 0.000, C 0.000 }
gfCNCPoint3[8006] = {X 335.3381, Y 89.9147, Z -3.8333, A 0.000, B 0.000, C 0.000 }
gfCNCPoint3[8007] = {X 339.4788, Y 90.2352, Z -3.8333, A 0.000, B 0.000, C 0.000 }
gfCNCPoint3[8008] = {X 343.6280, Y 90.4149, Z -3.8333, A 0.000, B 0.000, C 0.000 }
gfCNCPoint3[8009] = {X 347.7809, Y 90.4537, Z -3.8333, A 0.000, B 0.000, C 0.000 }
gfCNCPoint3[8010] = {X 352.1650, Y 90.4152, Z -3.8333, A 0.000, B 0.000, C 0.000 }
gfCNCPoint3[8011] = {X 356.5449, Y 90.2193, Z -3.8333, A 0.000, B 0.000, C 0.000 }
gfCNCPoint3[8012] = {X 360.9150, Y 89.8660, Z -3.8333, A 0.000, B 0.000, C 0.000 }
gfCNCPoint3[8013] = {X 363.2338, Y 89.5776, Z -3.8333, A 0.000, B 0.000, C 0.000 }
gfCNCPoint3[8014] = {X 365.5310, Y 89.1503, Z -3.8333, A 0.000, B 0.000, C 0.000 }
gfCNCPoint3[8015] = {X 367.7985, Y 88.5858, Z -3.8333, A 0.000, B 0.000, C 0.000 }
gfCNCPoint3[8016] = {X 368.7388, Y 88.2697, Z -3.8333, A 0.000, B 0.000, C 0.000 }
gfCNCPoint3[8017] = {X 369.6378, Y 87.8501, Z -3.8333, A 0.000, B 0.000, C 0.000 }
gfCNCPoint3[8018] = {X 370.4840, Y 87.3323, Z -3.8333, A 0.000, B 0.000, C 0.000 }
gfCNCPoint3[8019] = {X 370.6559, Y 87.1534, Z -3.8333, A 0.000, B 0.000, C 0.000 }
gfCNCPoint3[8020] = {X 370.7445, Y 86.9218, Z -3.8333, A 0.000, B 0.000, C 0.000 }
gfCNCPoint3[8021] = {X 370.9364, Y 85.3802, Z -3.8333, A 0.000, B 0.000, C 0.000 }
gfCNCPoint3[8022] = {X 371.0004, Y 83.8281, Z -3.8333, A 0.000, B 0.000, C 0.000 }
gfCNCPoint3[8023] = {X 371.0006, Y 63.1422, Z -3.8333, A 0.000, B 0.000, C 0.000 }
gfCNCPoint3[8024] = {X 370.1520, Y 62.9476, Z -3.8333, A 0.000, B 0.000, C 0.000 }
gfCNCPoint3[8025] = {X 369.3611, Y 62.5837, Z -3.8333, A 0.000, B 0.000, C 0.000 }
gfCNCPoint3[8026] = {X 368.6611, Y 62.0659, Z -3.8333, A 0.000, B 0.000, C 0.000 }
gfCNCPoint3[8027] = {X 368.0817, Y 61.4161, Z -3.8333, A 0.000, B 0.000, C 0.000 }
gfCNCPoint3[8028] = {X 367.6472, Y 60.6617, Z -3.8333, A 0.000, B 0.000, C 0.000 }
gfCNCPoint3[8029] = {X 367.3760, Y 59.8343, Z -3.8333, A 0.000, B 0.000, C 0.000 }
gfCNCPoint3[8030] = {X 367.2794, Y 58.9691, Z -3.8333, A 0.000, B 0.000, C 0.000 }
gfCNCPoint3[8031] = {X 367.2793, Y 58.0000, Z -3.8333, A 0.000, B 0.000, C 0.000 }
gfCNCPoint3[8032] = {X 367.3856, Y 57.0565, Z -3.8333, A 0.000, B 0.000, C 0.000 }
gfCNCPoint3[8033] = {X 367.6992, Y 56.1603, Z -3.8333, A 0.000, B 0.000, C 0.000 }
gfCNCPoint3[8034] = {X 368.2043, Y 55.3564, Z -3.8333, A 0.000, B 0.000, C 0.000 }
gfCNCPoint3[8035] = {X 368.8757, Y 54.6850, Z -3.8333, A 0.000, B 0.000, C 0.000 }
gfCNCPoint3[8036] = {X 369.6796, Y 54.1799, Z -3.8333, A 0.000, B 0.000, C 0.000 }
gfCNCPoint3[8037] = {X 370.5758, Y 53.8663, Z -3.8333, A 0.000, B 0.000, C 0.000 }
gfCNCPoint3[8038] = {X 371.5193, Y 53.7600, Z -3.8333, A 0.000, B 0.000, C 0.000 }
gfCNCPoint3[8039] = {X 388.0597, Y 53.7600, Z -3.8333, A 0.000, B 0.000, C 0.000 }
gfCNCPoint3[8040] = {X 389.0032, Y 53.8663, Z -3.8333, A 0.000, B 0.000, C 0.000 }
gfCNCPoint3[8041] = {X 389.8993, Y 54.1799, Z -3.8333, A 0.000, B 0.000, C 0.000 }
gfCNCPoint3[8042] = {X 390.7033, Y 54.6850, Z -3.8333, A 0.000, B 0.000, C 0.000 }
gfCNCPoint3[8043] = {X 391.3746, Y 55.3564, Z -3.8333, A 0.000, B 0.000, C 0.000 }
gfCNCPoint3[8044] = {X 391.8798, Y 56.1603, Z -3.8333, A 0.000, B 0.000, C 0.000 }
gfCNCPoint3[8045] = {X 392.1934, Y 57.0565, Z -3.8333, A 0.000, B 0.000, C 0.000 }
gfCNCPoint3[8046] = {X 392.2997, Y 58.0000, Z -3.8333, A 0.000, B 0.000, C 0.000 }
gfCNCPoint3[8047] = {X 392.2997, Y 58.9342, Z -3.8333, A 0.000, B 0.000, C 0.000 }
gfCNCPoint3[8048] = {X 392.1873, Y 59.9036, Z -3.8333, A 0.000, B 0.000, C 0.000 }
gfCNCPoint3[8049] = {X 391.8563, Y 60.8217, Z -3.8333, A 0.000, B 0.000, C 0.000 }
gfCNCPoint3[8050] = {X 391.4128, Y 61.5313, Z -3.8333, A 0.000, B 0.000, C 0.000 }
gfCNCPoint3[8051] = {X 390.8392, Y 62.1406, Z -3.8333, A 0.000, B 0.000, C 0.000 }
gfCNCPoint3[8052] = {X 390.1576, Y 62.6260, Z -3.8333, A 0.000, B 0.000, C 0.000 }
gfCNCPoint3[8053] = {X 389.3943, Y 62.9689, Z -3.8333, A 0.000, B 0.000, C 0.000 }
gfCNCPoint3[8054] = {X 388.5786, Y 63.1561, Z -3.8333, A 0.000, B 0.000, C 0.000 }
gfCNCPoint3[8055] = {X 388.5766, Y 84.6151, Z -3.8333, A 0.000, B 0.000, C 0.000 }
gfCNCPoint3[8056] = {X 388.5170, Y 86.2666, Z -3.8333, A 0.000, B 0.000, C 0.000 }
gfCNCPoint3[8057] = {X 388.3135, Y 87.9065, Z -3.8333, A 0.000, B 0.000, C 0.000 }
gfCNCPoint3[8058] = {X 387.9677, Y 89.5225, Z -3.8333, A 0.000, B 0.000, C 0.000 }
gfCNCPoint3[8059] = {X 387.4391, Y 91.0992, Z -3.8333, A 0.000, B 0.000, C 0.000 }
gfCNCPoint3[8060] = {X 386.6946, Y 92.5861, Z -3.8333, A 0.000, B 0.000, C 0.000 }
gfCNCPoint3[8061] = {X 385.7489, Y 93.9539, Z -3.8333, A 0.000, B 0.000, C 0.000 }
gfCNCPoint3[8062] = {X 384.6207, Y 95.1755, Z -3.8333, A 0.000, B 0.000, C 0.000 }
gfCNCPoint3[8063] = {X 383.1129, Y 96.4459, Z -3.8333, A 0.000, B 0.000, C 0.000 }
gfCNCPoint3[8064] = {X 381.4787, Y 97.5491, Z -3.8333, A 0.000, B 0.000, C 0.000 }
gfCNCPoint3[8065] = {X 379.7367, Y 98.4727, Z -3.8333, A 0.000, B 0.000, C 0.000 }
gfCNCPoint3[8066] = {X 377.4708, Y 99.4266, Z -3.8333, A 0.000, B 0.000, C 0.000 }
gfCNCPoint3[8067] = {X 375.1422, Y 100.2150, Z -3.8333, A 0.000, B 0.000, C 0.000 }
gfCNCPoint3[8068] = {X 372.7628, Y 100.8339, Z -3.8333, A 0.000, B 0.000, C 0.000 }
gfCNCPoint3[8069] = {X 368.9550, Y 101.5705, Z -3.8333, A 0.000, B 0.000, C 0.000 }
gfCNCPoint3[8070] = {X 365.1161, Y 102.1233, Z -3.8333, A 0.000, B 0.000, C 0.000 }
gfCNCPoint3[8071] = {X 361.2551, Y 102.4909, Z -3.8333, A 0.000, B 0.000, C 0.000 }
gfCNCPoint3[8072] = {X 357.2499, Y 102.7315, Z -3.8333, A 0.000, B 0.000, C 0.000 }
gfCNCPoint3[8073] = {X 353.2403, Y 102.8849, Z -3.8333, A 0.000, B 0.000, C 0.000 }
gfCNCPoint3[8074] = {X 353.3498, Y 106.8834, Z -3.8333, A 0.000, B 0.000, C 0.000 }
gfCNCPoint3[8075] = {X 353.2381, Y 102.8049, Z -3.8333, A 0.000, B 0.000, C 0.000 }
gfCNCPoint3[8076] = {X 347.7206, Y 102.8734, Z -3.8333, A 0.000, B 0.000, C 0.000 }
gfCNCPoint3[8077] = {X 342.2035, Y 102.7767, Z -3.8333, A 0.000, B 0.000, C 0.000 }
gfCNCPoint3[8078] = {X 336.6917, Y 102.5151, Z -3.8333, A 0.000, B 0.000, C 0.000 }
gfCNCPoint3[8079] = {X 333.2080, Y 102.2393, Z -3.8333, A 0.000, B 0.000, C 0.000 }
gfCNCPoint3[8080] = {X 329.7379, Y 101.8271, Z -3.8333, A 0.000, B 0.000, C 0.000 }
gfCNCPoint3[8081] = {X 326.2865, Y 101.2791, Z -3.8333, A 0.000, B 0.000, C 0.000 }
gfCNCPoint3[8082] = {X 323.4481, Y 100.6778, Z -3.8333, A 0.000, B 0.000, C 0.000 }
gfCNCPoint3[8083] = {X 320.6619, Y 99.8681, Z -3.8333, A 0.000, B 0.000, C 0.000 }
gfCNCPoint3[8084] = {X 317.9433, Y 98.8544, Z -3.8333, A 0.000, B 0.000, C 0.000 }
gfCNCPoint3[8085] = {X 316.4429, Y 98.1615, Z -3.8333, A 0.000, B 0.000, C 0.000 }
gfCNCPoint3[8086] = {X 315.0054, Y 97.3460, Z -3.8333, A 0.000, B 0.000, C 0.000 }
gfCNCPoint3[8087] = {X 313.6408, Y 96.4137, Z -3.8333, A 0.000, B 0.000, C 0.000 }
gfCNCPoint3[8088] = {X 312.3587, Y 95.3709, Z -3.8333, A 0.000, B 0.000, C 0.000 }
gfCNCPoint3[8089] = {X 311.3684, Y 94.3859, Z -3.8333, A 0.000, B 0.000, C 0.000 }
gfCNCPoint3[8090] = {X 310.5019, Y 93.2905, Z -3.8333, A 0.000, B 0.000, C 0.000 }
gfCNCPoint3[8091] = {X 309.7714, Y 92.1000, Z -3.8333, A 0.000, B 0.000, C 0.000 }
gfCNCPoint3[8092] = {X 309.1873, Y 90.8312, Z -3.8333, A 0.000, B 0.000, C 0.000 }
gfCNCPoint3[8093] = {X 308.7579, Y 89.5022, Z -3.8333, A 0.000, B 0.000, C 0.000 }
gfCNCPoint3[8094] = {X 308.4173, Y 87.8925, Z -3.8333, A 0.000, B 0.000, C 0.000 }
gfCNCPoint3[8095] = {X 308.2161, Y 86.2595, Z -3.8333, A 0.000, B 0.000, C 0.000 }
gfCNCPoint3[8096] = {X 308.1557, Y 84.6153, Z -3.8333, A 0.000, B 0.000, C 0.000 }
gfCNCPoint3[8097] = {X 308.1570, Y 63.0708, Z -3.8333, A 0.000, B 0.000, C 0.000 }
gfCNCPoint3[8098] = {X 307.3118, Y 62.8908, Z -3.8333, A 0.000, B 0.000, C 0.000 }
gfCNCPoint3[8099] = {X 306.5220, Y 62.5401, Z -3.8333, A 0.000, B 0.000, C 0.000 }
gfCNCPoint3[8100] = {X 305.8218, Y 62.0337, Z -3.8333, A 0.000, B 0.000, C 0.000 }
gfCNCPoint3[8101] = {X 305.2412, Y 61.3937, Z -3.8333, A 0.000, B 0.000, C 0.000 }
gfCNCPoint3[8102] = {X 304.8055, Y 60.6475, Z -3.8333, A 0.000, B 0.000, C 0.000 }
gfCNCPoint3[8103] = {X 304.5333, Y 59.8273, Z -3.8333, A 0.000, B 0.000, C 0.000 }
gfCNCPoint3[8104] = {X 304.4364, Y 58.9686, Z -3.8333, A 0.000, B 0.000, C 0.000 }
gfCNCPoint3[8105] = {X 304.4362, Y 58.0000, Z -3.8333, A 0.000, B 0.000, C 0.000 }
gfCNCPoint3[8106] = {X 304.5405, Y 57.0743, Z -3.8333, A 0.000, B 0.000, C 0.000 }
gfCNCPoint3[8107] = {X 304.8482, Y 56.1950, Z -3.8333, A 0.000, B 0.000, C 0.000 }
gfCNCPoint3[8108] = {X 305.3438, Y 55.4063, Z -3.8333, A 0.000, B 0.000, C 0.000 }
gfCNCPoint3[8109] = {X 306.0025, Y 54.7476, Z -3.8333, A 0.000, B 0.000, C 0.000 }
gfCNCPoint3[8110] = {X 306.7913, Y 54.2520, Z -3.8333, A 0.000, B 0.000, C 0.000 }
gfCNCPoint3[8111] = {X 307.6705, Y 53.9443, Z -3.8333, A 0.000, B 0.000, C 0.000 }
gfCNCPoint3[8112] = {X 308.5962, Y 53.8400, Z -3.8333, A 0.000, B 0.000, C 0.000 }
gfCNCPoint3[8113] = {X 324.3107, Y 53.8400, Z -3.8333, A 0.000, B 0.000, C 0.000 }
gfCNCPoint3[8114] = {X 325.2364, Y 53.9443, Z -3.8333, A 0.000, B 0.000, C 0.000 }
gfCNCPoint3[8115] = {X 326.1156, Y 54.2520, Z -3.8333, A 0.000, B 0.000, C 0.000 }
gfCNCPoint3[8116] = {X 326.9044, Y 54.7476, Z -3.8333, A 0.000, B 0.000, C 0.000 }
gfCNCPoint3[8117] = {X 327.5631, Y 55.4063, Z -3.8333, A 0.000, B 0.000, C 0.000 }
gfCNCPoint3[8118] = {X 328.0587, Y 56.1950, Z -3.8333, A 0.000, B 0.000, C 0.000 }
gfCNCPoint3[8119] = {X 328.3664, Y 57.0743, Z -3.8333, A 0.000, B 0.000, C 0.000 }
gfCNCPoint3[8120] = {X 328.4707, Y 58.0000, Z -3.8333, A 0.000, B 0.000, C 0.000 }
gfCNCPoint3[8121] = {X 328.4707, Y 58.9350, Z -3.8333, A 0.000, B 0.000, C 0.000 }
gfCNCPoint3[8122] = {X 328.3758, Y 59.7983, Z -3.8333, A 0.000, B 0.000, C 0.000 }
gfCNCPoint3[8123] = {X 328.1053, Y 60.6237, Z -3.8333, A 0.000, B 0.000, C 0.000 }
gfCNCPoint3[8124] = {X 327.6708, Y 61.3757, Z -3.8333, A 0.000, B 0.000, C 0.000 }
gfCNCPoint3[8125] = {X 327.0909, Y 62.0222, Z -3.8333, A 0.000, B 0.000, C 0.000 }
gfCNCPoint3[8126] = {X 326.3904, Y 62.5356, Z -3.8333, A 0.000, B 0.000, C 0.000 }
gfCNCPoint3[8127] = {X 325.5993, Y 62.8939, Z -3.8333, A 0.000, B 0.000, C 0.000 }
gfCNCPoint3[8128] = {X 324.7513, Y 63.0818, Z -3.8333, A 0.000, B 0.000, C 0.000 }
gfCNCPoint3[8129] = {X 324.7529, Y 83.2304, Z -3.8333, A 0.000, B 0.000, C 0.000 }
gfCNCPoint3[8130] = {X 324.7664, Y 84.6153, Z -3.8333, A 0.000, B 0.000, C 0.000 }
gfCNCPoint3[8131] = {X 324.8468, Y 85.8843, Z -3.8333, A 0.000, B 0.000, C 0.000 }
gfCNCPoint3[8132] = {X 325.0779, Y 87.1347, Z -3.8333, A 0.000, B 0.000, C 0.000 }
gfCNCPoint3[8133] = {X 325.3539, Y 87.4461, Z -3.8333, A 0.000, B 0.000, C 0.000 }
gfCNCPoint3[8134] = {X 325.6979, Y 87.6801, Z -3.8333, A 0.000, B 0.000, C 0.000 }
gfCNCPoint3[8135] = {X 326.1501, Y 87.9356, Z -3.8333, A 0.000, B 0.000, C 0.000 }
gfCNCPoint3[8136] = {X 327.6066, Y 88.5406, Z -3.8333, A 0.000, B 0.000, C 0.000 }
gfCNCPoint3[8137] = {X 329.1206, Y 88.9822, Z -3.8333, A 0.000, B 0.000, C 0.000 }
gfCNCPoint3[8138] = {X 332.2076, Y 89.6002, Z -3.8333, A 0.000, B 0.000, C 0.000 }
gfCNCPoint3[8139] = {X 335.3310, Y 89.9944, Z -3.8333, A 0.000, B 0.000, C 0.000 }
gfCNCPoint3[8140] = {X 339.4743, Y 90.3150, Z -3.8333, A 0.000, B 0.000, C 0.000 }
gfCNCPoint3[8141] = {X 343.6260, Y 90.4949, Z -3.8333, A 0.000, B 0.000, C 0.000 }
gfCNCPoint3[8142] = {X 347.7815, Y 90.5337, Z -3.8333, A 0.000, B 0.000, C 0.000 }
gfCNCPoint3[8143] = {X 352.1681, Y 90.4952, Z -3.8333, A 0.000, B 0.000, C 0.000 }
gfCNCPoint3[8144] = {X 356.5504, Y 90.2991, Z -3.8333, A 0.000, B 0.000, C 0.000 }
gfCNCPoint3[8145] = {X 360.9228, Y 89.9456, Z -3.8333, A 0.000, B 0.000, C 0.000 }
gfCNCPoint3[8146] = {X 363.2463, Y 89.6566, Z -3.8333, A 0.000, B 0.000, C 0.000 }
gfCNCPoint3[8147] = {X 365.5481, Y 89.2285, Z -3.8333, A 0.000, B 0.000, C 0.000 }
gfCNCPoint3[8148] = {X 367.8201, Y 88.6628, Z -3.8333, A 0.000, B 0.000, C 0.000 }
gfCNCPoint3[8149] = {X 368.7688, Y 88.3438, Z -3.8333, A 0.000, B 0.000, C 0.000 }
gfCNCPoint3[8150] = {X 369.6758, Y 87.9205, Z -3.8333, A 0.000, B 0.000, C 0.000 }
gfCNCPoint3[8151] = {X 370.5295, Y 87.3981, Z -3.8333, A 0.000, B 0.000, C 0.000 }
gfCNCPoint3[8152] = {X 370.7234, Y 87.1963, Z -3.8333, A 0.000, B 0.000, C 0.000 }
gfCNCPoint3[8153] = {X 370.8234, Y 86.9349, Z -3.8333, A 0.000, B 0.000, C 0.000 }
gfCNCPoint3[8154] = {X 371.0161, Y 85.3868, Z -3.8333, A 0.000, B 0.000, C 0.000 }
gfCNCPoint3[8155] = {X 371.0804, Y 83.8281, Z -3.8333, A 0.000, B 0.000, C 0.000 }
gfCNCPoint3[8156] = {X 371.0806, Y 63.0709, Z -3.8333, A 0.000, B 0.000, C 0.000 }
gfCNCPoint3[8157] = {X 370.9782, Y 63.0587, Z -3.8333, A 0.000, B 0.000, C 0.000 }
gfCNCPoint3[8158] = {X 370.8760, Y 63.0440, Z -3.8333, A 0.000, B 0.000, C 0.000 }
gfCNCPoint3[8159] = {X 369.9385, Y 62.7820, Z -3.8333, A 0.000, B 0.000, C 0.000 }
gfCNCPoint3[8160] = {X 369.0875, Y 62.3093, Z -3.8333, A 0.000, B 0.000, C 0.000 }
gfCNCPoint3[8161] = {X 368.3697, Y 61.6517, Z -3.8333, A 0.000, B 0.000, C 0.000 }
gfCNCPoint3[8162] = {X 367.8243, Y 60.8453, Z -3.8333, A 0.000, B 0.000, C 0.000 }
gfCNCPoint3[8163] = {X 367.4813, Y 59.9342, Z -3.8333, A 0.000, B 0.000, C 0.000 }
gfCNCPoint3[8164] = {X 367.3594, Y 58.9684, Z -3.8333, A 0.000, B 0.000, C 0.000 }
gfCNCPoint3[8165] = {X 367.3593, Y 58.0000, Z -3.8333, A 0.000, B 0.000, C 0.000 }
gfCNCPoint3[8166] = {X 367.4636, Y 57.0743, Z -3.8333, A 0.000, B 0.000, C 0.000 }
gfCNCPoint3[8167] = {X 367.7713, Y 56.1950, Z -3.8333, A 0.000, B 0.000, C 0.000 }
gfCNCPoint3[8168] = {X 368.2669, Y 55.4063, Z -3.8333, A 0.000, B 0.000, C 0.000 }
gfCNCPoint3[8169] = {X 368.9256, Y 54.7476, Z -3.8333, A 0.000, B 0.000, C 0.000 }
gfCNCPoint3[8170] = {X 369.7143, Y 54.2520, Z -3.8333, A 0.000, B 0.000, C 0.000 }
gfCNCPoint3[8171] = {X 370.5936, Y 53.9443, Z -3.8333, A 0.000, B 0.000, C 0.000 }
gfCNCPoint3[8172] = {X 371.5193, Y 53.8400, Z -3.8333, A 0.000, B 0.000, C 0.000 }
gfCNCPoint3[8173] = {X 388.0597, Y 53.8400, Z -3.8333, A 0.000, B 0.000, C 0.000 }
gfCNCPoint3[8174] = {X 388.9854, Y 53.9443, Z -3.8333, A 0.000, B 0.000, C 0.000 }
gfCNCPoint3[8175] = {X 389.8646, Y 54.2520, Z -3.8333, A 0.000, B 0.000, C 0.000 }
gfCNCPoint3[8176] = {X 390.6534, Y 54.7476, Z -3.8333, A 0.000, B 0.000, C 0.000 }
gfCNCPoint3[8177] = {X 391.3121, Y 55.4063, Z -3.8333, A 0.000, B 0.000, C 0.000 }
gfCNCPoint3[8178] = {X 391.8077, Y 56.1950, Z -3.8333, A 0.000, B 0.000, C 0.000 }
gfCNCPoint3[8179] = {X 392.1154, Y 57.0743, Z -3.8333, A 0.000, B 0.000, C 0.000 }
gfCNCPoint3[8180] = {X 392.2197, Y 58.0000, Z -3.8333, A 0.000, B 0.000, C 0.000 }
gfCNCPoint3[8181] = {X 392.2197, Y 58.9342, Z -3.8333, A 0.000, B 0.000, C 0.000 }
gfCNCPoint3[8182] = {X 392.1095, Y 59.8853, Z -3.8333, A 0.000, B 0.000, C 0.000 }
gfCNCPoint3[8183] = {X 391.7847, Y 60.7860, Z -3.8333, A 0.000, B 0.000, C 0.000 }
gfCNCPoint3[8184] = {X 391.2411, Y 61.6154, Z -3.8333, A 0.000, B 0.000, C 0.000 }
gfCNCPoint3[8185] = {X 390.5174, Y 62.2934, Z -3.8333, A 0.000, B 0.000, C 0.000 }
gfCNCPoint3[8186] = {X 389.6545, Y 62.7820, Z -3.8333, A 0.000, B 0.000, C 0.000 }
gfCNCPoint3[8187] = {X 388.7007, Y 63.0537, Z -3.8333, A 0.000, B 0.000, C 0.000 }
gfCNCPoint3[8188] = {X 388.6005, Y 63.0685, Z -3.8333, A 0.000, B 0.000, C 0.000 }
gfCNCPoint3[8189] = {X 388.4999, Y 63.0808, Z -3.8333, A 0.000, B 0.000, C 0.000 }
gfCNCPoint3[8190] = {X 388.4966, Y 84.6154, Z -3.8333, A 0.000, B 0.000, C 0.000 }
gfCNCPoint3[8191] = {X 388.4372, Y 86.2600, Z -3.8333, A 0.000, B 0.000, C 0.000 }
gfCNCPoint3[8192] = {X 388.2346, Y 87.8931, Z -3.8333, A 0.000, B 0.000, C 0.000 }
gfCNCPoint3[8193] = {X 387.8903, Y 89.5024, Z -3.8333, A 0.000, B 0.000, C 0.000 }
gfCNCPoint3[8194] = {X 387.3653, Y 91.0684, Z -3.8333, A 0.000, B 0.000, C 0.000 }
gfCNCPoint3[8195] = {X 386.6258, Y 92.5453, Z -3.8333, A 0.000, B 0.000, C 0.000 }
gfCNCPoint3[8196] = {X 385.6865, Y 93.9039, Z -3.8333, A 0.000, B 0.000, C 0.000 }
gfCNCPoint3[8197] = {X 384.5659, Y 95.1172, Z -3.8333, A 0.000, B 0.000, C 0.000 }
gfCNCPoint3[8198] = {X 383.0646, Y 96.3821, Z -3.8333, A 0.000, B 0.000, C 0.000 }
gfCNCPoint3[8199] = {X 381.4375, Y 97.4806, Z -3.8333, A 0.000, B 0.000, C 0.000 }
gfCNCPoint3[8200] = {X 379.7030, Y 98.4001, Z -3.8333, A 0.000, B 0.000, C 0.000 }
gfCNCPoint3[8201] = {X 377.4424, Y 99.3518, Z -3.8333, A 0.000, B 0.000, C 0.000 }
gfCNCPoint3[8202] = {X 375.1192, Y 100.1383, Z -3.8333, A 0.000, B 0.000, C 0.000 }
gfCNCPoint3[8203] = {X 372.7455, Y 100.7558, Z -3.8333, A 0.000, B 0.000, C 0.000 }
gfCNCPoint3[8204] = {X 368.9415, Y 101.4917, Z -3.8333, A 0.000, B 0.000, C 0.000 }
gfCNCPoint3[8205] = {X 365.1066, Y 102.0439, Z -3.8333, A 0.000, B 0.000, C 0.000 }
gfCNCPoint3[8206] = {X 361.2495, Y 102.4111, Z -3.8333, A 0.000, B 0.000, C 0.000 }
gfCNCPoint3[8207] = {X 357.2459, Y 102.6516, Z -3.8333, A 0.000, B 0.000, C 0.000 }
gfCNCPoint3[8208] = {X 353.2381, Y 102.8049, Z -3.8333, A 0.000, B 0.000, C 0.000 }
gfCNCPoint3[8209] = {X 353.3476, Y 106.8034, Z -3.8333, A 0.000, B 0.000, C 0.000 }
gfCNCPoint3[8210] = {X 353.2360, Y 102.7250, Z -3.8333, A 0.000, B 0.000, C 0.000 }
gfCNCPoint3[8211] = {X 347.7208, Y 102.7934, Z -3.8333, A 0.000, B 0.000, C 0.000 }
gfCNCPoint3[8212] = {X 342.2061, Y 102.6968, Z -3.8333, A 0.000, B 0.000, C 0.000 }
gfCNCPoint3[8213] = {X 336.6967, Y 102.4352, Z -3.8333, A 0.000, B 0.000, C 0.000 }
gfCNCPoint3[8214] = {X 333.2160, Y 102.1597, Z -3.8333, A 0.000, B 0.000, C 0.000 }
gfCNCPoint3[8215] = {X 329.7488, Y 101.7479, Z -3.8333, A 0.000, B 0.000, C 0.000 }
gfCNCPoint3[8216] = {X 326.3005, Y 101.2003, Z -3.8333, A 0.000, B 0.000, C 0.000 }
gfCNCPoint3[8217] = {X 323.4677, Y 100.6002, Z -3.8333, A 0.000, B 0.000, C 0.000 }
gfCNCPoint3[8218] = {X 320.6871, Y 99.7921, Z -3.8333, A 0.000, B 0.000, C 0.000 }
gfCNCPoint3[8219] = {X 317.9740, Y 98.7805, Z -3.8333, A 0.000, B 0.000, C 0.000 }
gfCNCPoint3[8220] = {X 316.4795, Y 98.0904, Z -3.8333, A 0.000, B 0.000, C 0.000 }
gfCNCPoint3[8221] = {X 315.0478, Y 97.2782, Z -3.8333, A 0.000, B 0.000, C 0.000 }
gfCNCPoint3[8222] = {X 313.6887, Y 96.3496, Z -3.8333, A 0.000, B 0.000, C 0.000 }
gfCNCPoint3[8223] = {X 312.4117, Y 95.3110, Z -3.8333, A 0.000, B 0.000, C 0.000 }
gfCNCPoint3[8224] = {X 311.4281, Y 94.3327, Z -3.8333, A 0.000, B 0.000, C 0.000 }
gfCNCPoint3[8225] = {X 310.5675, Y 93.2447, Z -3.8333, A 0.000, B 0.000, C 0.000 }
gfCNCPoint3[8226] = {X 309.8420, Y 92.0623, Z -3.8333, A 0.000, B 0.000, C 0.000 }
gfCNCPoint3[8227] = {X 309.2619, Y 90.8022, Z -3.8333, A 0.000, B 0.000, C 0.000 }
gfCNCPoint3[8228] = {X 308.8353, Y 89.4822, Z -3.8333, A 0.000, B 0.000, C 0.000 }
gfCNCPoint3[8229] = {X 308.4961, Y 87.8792, Z -3.8333, A 0.000, B 0.000, C 0.000 }
gfCNCPoint3[8230] = {X 308.2958, Y 86.2530, Z -3.8333, A 0.000, B 0.000, C 0.000 }
gfCNCPoint3[8231] = {X 308.2357, Y 84.6156, Z -3.8333, A 0.000, B 0.000, C 0.000 }
gfCNCPoint3[8232] = {X 308.2370, Y 62.9982, Z -3.8333, A 0.000, B 0.000, C 0.000 }
gfCNCPoint3[8233] = {X 307.3952, Y 62.8333, Z -3.8333, A 0.000, B 0.000, C 0.000 }
gfCNCPoint3[8234] = {X 306.6066, Y 62.4961, Z -3.8333, A 0.000, B 0.000, C 0.000 }
gfCNCPoint3[8235] = {X 305.9059, Y 62.0014, Z -3.8333, A 0.000, B 0.000, C 0.000 }
gfCNCPoint3[8236] = {X 305.3241, Y 61.3711, Z -3.8333, A 0.000, B 0.000, C 0.000 }
gfCNCPoint3[8237] = {X 304.8869, Y 60.6332, Z -3.8333, A 0.000, B 0.000, C 0.000 }
gfCNCPoint3[8238] = {X 304.6136, Y 59.8202, Z -3.8333, A 0.000, B 0.000, C 0.000 }
gfCNCPoint3[8239] = {X 304.5164, Y 58.9680, Z -3.8333, A 0.000, B 0.000, C 0.000 }
gfCNCPoint3[8240] = {X 304.5162, Y 58.0000, Z -3.8333, A 0.000, B 0.000, C 0.000 }
gfCNCPoint3[8241] = {X 304.6185, Y 57.0921, Z -3.8333, A 0.000, B 0.000, C 0.000 }
gfCNCPoint3[8242] = {X 304.9203, Y 56.2298, Z -3.8333, A 0.000, B 0.000, C 0.000 }
gfCNCPoint3[8243] = {X 305.4064, Y 55.4562, Z -3.8333, A 0.000, B 0.000, C 0.000 }
gfCNCPoint3[8244] = {X 306.0524, Y 54.8101, Z -3.8333, A 0.000, B 0.000, C 0.000 }
gfCNCPoint3[8245] = {X 306.8260, Y 54.3240, Z -3.8333, A 0.000, B 0.000, C 0.000 }
gfCNCPoint3[8246] = {X 307.6883, Y 54.0223, Z -3.8333, A 0.000, B 0.000, C 0.000 }
gfCNCPoint3[8247] = {X 308.5962, Y 53.9200, Z -3.8333, A 0.000, B 0.000, C 0.000 }
gfCNCPoint3[8248] = {X 324.3107, Y 53.9200, Z -3.8333, A 0.000, B 0.000, C 0.000 }
gfCNCPoint3[8249] = {X 325.2186, Y 54.0223, Z -3.8333, A 0.000, B 0.000, C 0.000 }
gfCNCPoint3[8250] = {X 326.0809, Y 54.3240, Z -3.8333, A 0.000, B 0.000, C 0.000 }
gfCNCPoint3[8251] = {X 326.8545, Y 54.8101, Z -3.8333, A 0.000, B 0.000, C 0.000 }
gfCNCPoint3[8252] = {X 327.5006, Y 55.4562, Z -3.8333, A 0.000, B 0.000, C 0.000 }
gfCNCPoint3[8253] = {X 327.9866, Y 56.2298, Z -3.8333, A 0.000, B 0.000, C 0.000 }
gfCNCPoint3[8254] = {X 328.2884, Y 57.0921, Z -3.8333, A 0.000, B 0.000, C 0.000 }
gfCNCPoint3[8255] = {X 328.3907, Y 58.0000, Z -3.8333, A 0.000, B 0.000, C 0.000 }
gfCNCPoint3[8256] = {X 328.3907, Y 58.9346, Z -3.8333, A 0.000, B 0.000, C 0.000 }
gfCNCPoint3[8257] = {X 328.2954, Y 59.7914, Z -3.8333, A 0.000, B 0.000, C 0.000 }
gfCNCPoint3[8258] = {X 328.0239, Y 60.6096, Z -3.8333, A 0.000, B 0.000, C 0.000 }
gfCNCPoint3[8259] = {X 327.5881, Y 61.3534, Z -3.8333, A 0.000, B 0.000, C 0.000 }
gfCNCPoint3[8260] = {X 327.0069, Y 61.9901, Z -3.8333, A 0.000, B 0.000, C 0.000 }
gfCNCPoint3[8261] = {X 326.3059, Y 62.4920, Z -3.8333, A 0.000, B 0.000, C 0.000 }
gfCNCPoint3[8262] = {X 325.5159, Y 62.8369, Z -3.8333, A 0.000, B 0.000, C 0.000 }
gfCNCPoint3[8263] = {X 324.6713, Y 63.0099, Z -3.8333, A 0.000, B 0.000, C 0.000 }
gfCNCPoint3[8264] = {X 324.6729, Y 83.2308, Z -3.8333, A 0.000, B 0.000, C 0.000 }
gfCNCPoint3[8265] = {X 324.6864, Y 84.6156, Z -3.8333, A 0.000, B 0.000, C 0.000 }
gfCNCPoint3[8266] = {X 324.7683, Y 85.9013, Z -3.8333, A 0.000, B 0.000, C 0.000 }
gfCNCPoint3[8267] = {X 325.0037, Y 87.1679, Z -3.8333, A 0.000, B 0.000, C 0.000 }
gfCNCPoint3[8268] = {X 325.2949, Y 87.5007, Z -3.8333, A 0.000, B 0.000, C 0.000 }
gfCNCPoint3[8269] = {X 325.6599, Y 87.7506, Z -3.8333, A 0.000, B 0.000, C 0.000 }
gfCNCPoint3[8270] = {X 326.1130, Y 88.0065, Z -3.8333, A 0.000, B 0.000, C 0.000 }
gfCNCPoint3[8271] = {X 327.5788, Y 88.6156, Z -3.8333, A 0.000, B 0.000, C 0.000 }
gfCNCPoint3[8272] = {X 329.1025, Y 89.0601, Z -3.8333, A 0.000, B 0.000, C 0.000 }
gfCNCPoint3[8273] = {X 332.1949, Y 89.6792, Z -3.8333, A 0.000, B 0.000, C 0.000 }
gfCNCPoint3[8274] = {X 335.3238, Y 90.0741, Z -3.8333, A 0.000, B 0.000, C 0.000 }
gfCNCPoint3[8275] = {X 339.4695, Y 90.3949, Z -3.8333, A 0.000, B 0.000, C 0.000 }
gfCNCPoint3[8276] = {X 343.6236, Y 90.5748, Z -3.8333, A 0.000, B 0.000, C 0.000 }
gfCNCPoint3[8277] = {X 347.7815, Y 90.6137, Z -3.8333, A 0.000, B 0.000, C 0.000 }
gfCNCPoint3[8278] = {X 352.1706, Y 90.5751, Z -3.8333, A 0.000, B 0.000, C 0.000 }
gfCNCPoint3[8279] = {X 356.5556, Y 90.3789, Z -3.8333, A 0.000, B 0.000, C 0.000 }
gfCNCPoint3[8280] = {X 360.9307, Y 90.0252, Z -3.8333, A 0.000, B 0.000, C 0.000 }
gfCNCPoint3[8281] = {X 363.2588, Y 89.7356, Z -3.8333, A 0.000, B 0.000, C 0.000 }
gfCNCPoint3[8282] = {X 365.5653, Y 89.3066, Z -3.8333, A 0.000, B 0.000, C 0.000 }
gfCNCPoint3[8283] = {X 367.8418, Y 88.7398, Z -3.8333, A 0.000, B 0.000, C 0.000 }
gfCNCPoint3[8284] = {X 368.7988, Y 88.4180, Z -3.8333, A 0.000, B 0.000, C 0.000 }
gfCNCPoint3[8285] = {X 369.7138, Y 87.9909, Z -3.8333, A 0.000, B 0.000, C 0.000 }
gfCNCPoint3[8286] = {X 370.5751, Y 87.4639, Z -3.8333, A 0.000, B 0.000, C 0.000 }
gfCNCPoint3[8287] = {X 370.7910, Y 87.2392, Z -3.8333, A 0.000, B 0.000, C 0.000 }
gfCNCPoint3[8288] = {X 370.9023, Y 86.9481, Z -3.8333, A 0.000, B 0.000, C 0.000 }
gfCNCPoint3[8289] = {X 371.0958, Y 85.3934, Z -3.8333, A 0.000, B 0.000, C 0.000 }
gfCNCPoint3[8290] = {X 371.1604, Y 83.8281, Z -3.8333, A 0.000, B 0.000, C 0.000 }
gfCNCPoint3[8291] = {X 371.1606, Y 62.9983, Z -3.8333, A 0.000, B 0.000, C 0.000 }
gfCNCPoint3[8292] = {X 371.0242, Y 62.9839, Z -3.8333, A 0.000, B 0.000, C 0.000 }
gfCNCPoint3[8293] = {X 370.8884, Y 62.9650, Z -3.8333, A 0.000, B 0.000, C 0.000 }
gfCNCPoint3[8294] = {X 369.9689, Y 62.7080, Z -3.8333, A 0.000, B 0.000, C 0.000 }
gfCNCPoint3[8295] = {X 369.1342, Y 62.2443, Z -3.8333, A 0.000, B 0.000, C 0.000 }
gfCNCPoint3[8296] = {X 368.4302, Y 61.5994, Z -3.8333, A 0.000, B 0.000, C 0.000 }
gfCNCPoint3[8297] = {X 367.8954, Y 60.8085, Z -3.8333, A 0.000, B 0.000, C 0.000 }
gfCNCPoint3[8298] = {X 367.5590, Y 59.9150, Z -3.8333, A 0.000, B 0.000, C 0.000 }
gfCNCPoint3[8299] = {X 367.4394, Y 58.9678, Z -3.8333, A 0.000, B 0.000, C 0.000 }
gfCNCPoint3[8300] = {X 367.4393, Y 58.0000, Z -3.8333, A 0.000, B 0.000, C 0.000 }
gfCNCPoint3[8301] = {X 367.5416, Y 57.0921, Z -3.8333, A 0.000, B 0.000, C 0.000 }
gfCNCPoint3[8302] = {X 367.8433, Y 56.2298, Z -3.8333, A 0.000, B 0.000, C 0.000 }
gfCNCPoint3[8303] = {X 368.3294, Y 55.4562, Z -3.8333, A 0.000, B 0.000, C 0.000 }
gfCNCPoint3[8304] = {X 368.9754, Y 54.8101, Z -3.8333, A 0.000, B 0.000, C 0.000 }
gfCNCPoint3[8305] = {X 369.7490, Y 54.3240, Z -3.8333, A 0.000, B 0.000, C 0.000 }
gfCNCPoint3[8306] = {X 370.6114, Y 54.0223, Z -3.8333, A 0.000, B 0.000, C 0.000 }
gfCNCPoint3[8307] = {X 371.5193, Y 53.9200, Z -3.8333, A 0.000, B 0.000, C 0.000 }
gfCNCPoint3[8308] = {X 388.0597, Y 53.9200, Z -3.8333, A 0.000, B 0.000, C 0.000 }
gfCNCPoint3[8309] = {X 388.9676, Y 54.0223, Z -3.8333, A 0.000, B 0.000, C 0.000 }
gfCNCPoint3[8310] = {X 389.8299, Y 54.3240, Z -3.8333, A 0.000, B 0.000, C 0.000 }
gfCNCPoint3[8311] = {X 390.6035, Y 54.8101, Z -3.8333, A 0.000, B 0.000, C 0.000 }
gfCNCPoint3[8312] = {X 391.2496, Y 55.4562, Z -3.8333, A 0.000, B 0.000, C 0.000 }
gfCNCPoint3[8313] = {X 391.7356, Y 56.2298, Z -3.8333, A 0.000, B 0.000, C 0.000 }
gfCNCPoint3[8314] = {X 392.0374, Y 57.0921, Z -3.8333, A 0.000, B 0.000, C 0.000 }
gfCNCPoint3[8315] = {X 392.1397, Y 58.0000, Z -3.8333, A 0.000, B 0.000, C 0.000 }
gfCNCPoint3[8316] = {X 392.1397, Y 58.9342, Z -3.8333, A 0.000, B 0.000, C 0.000 }
gfCNCPoint3[8317] = {X 392.0316, Y 59.8670, Z -3.8333, A 0.000, B 0.000, C 0.000 }
gfCNCPoint3[8318] = {X 391.7131, Y 60.7504, Z -3.8333, A 0.000, B 0.000, C 0.000 }
gfCNCPoint3[8319] = {X 391.1798, Y 61.5639, Z -3.8333, A 0.000, B 0.000, C 0.000 }
gfCNCPoint3[8320] = {X 390.4700, Y 62.2290, Z -3.8333, A 0.000, B 0.000, C 0.000 }
gfCNCPoint3[8321] = {X 389.6236, Y 62.7082, Z -3.8333, A 0.000, B 0.000, C 0.000 }
gfCNCPoint3[8322] = {X 388.6881, Y 62.9747, Z -3.8333, A 0.000, B 0.000, C 0.000 }
gfCNCPoint3[8323] = {X 388.5548, Y 62.9938, Z -3.8333, A 0.000, B 0.000, C 0.000 }
gfCNCPoint3[8324] = {X 388.4210, Y 63.0085, Z -3.8333, A 0.000, B 0.000, C 0.000 }
gfCNCPoint3[8325] = {X 388.4186, Y 63.1547, Z -3.8333, A 0.000, B 0.000, C 0.000 }
gfCNCPoint3[8326] = {X 388.4166, Y 84.6157, Z -3.8333, A 0.000, B 0.000, C 0.000 }
gfCNCPoint3[8327] = {X 388.3575, Y 86.2534, Z -3.8333, A 0.000, B 0.000, C 0.000 }
gfCNCPoint3[8328] = {X 388.1557, Y 87.8797, Z -3.8333, A 0.000, B 0.000, C 0.000 }
gfCNCPoint3[8329] = {X 387.8128, Y 89.4823, Z -3.8333, A 0.000, B 0.000, C 0.000 }
gfCNCPoint3[8330] = {X 387.2914, Y 91.0376, Z -3.8333, A 0.000, B 0.000, C 0.000 }
gfCNCPoint3[8331] = {X 386.5570, Y 92.5045, Z -3.8333, A 0.000, B 0.000, C 0.000 }
gfCNCPoint3[8332] = {X 385.6241, Y 93.8538, Z -3.8333, A 0.000, B 0.000, C 0.000 }
gfCNCPoint3[8333] = {X 384.5111, Y 95.0589, Z -3.8333, A 0.000, B 0.000, C 0.000 }
gfCNCPoint3[8334] = {X 383.0163, Y 96.3184, Z -3.8333, A 0.000, B 0.000, C 0.000 }
gfCNCPoint3[8335] = {X 381.3963, Y 97.4120, Z -3.8333, A 0.000, B 0.000, C 0.000 }
gfCNCPoint3[8336] = {X 379.6693, Y 98.3275, Z -3.8333, A 0.000, B 0.000, C 0.000 }
gfCNCPoint3[8337] = {X 377.4141, Y 99.2770, Z -3.8333, A 0.000, B 0.000, C 0.000 }
gfCNCPoint3[8338] = {X 375.0963, Y 100.0617, Z -3.8333, A 0.000, B 0.000, C 0.000 }
gfCNCPoint3[8339] = {X 372.7282, Y 100.6777, Z -3.8333, A 0.000, B 0.000, C 0.000 }
gfCNCPoint3[8340] = {X 368.9280, Y 101.4128, Z -3.8333, A 0.000, B 0.000, C 0.000 }
gfCNCPoint3[8341] = {X 365.0970, Y 101.9645, Z -3.8333, A 0.000, B 0.000, C 0.000 }
gfCNCPoint3[8342] = {X 361.2438, Y 102.3313, Z -3.8333, A 0.000, B 0.000, C 0.000 }
gfCNCPoint3[8343] = {X 357.2420, Y 102.5717, Z -3.8333, A 0.000, B 0.000, C 0.000 }
gfCNCPoint3[8344] = {X 353.2360, Y 102.7250, Z -3.8333, A 0.000, B 0.000, C 0.000 }
gfCNCPoint3[8345] = {X 353.3454, Y 106.7235, Z -3.8333, A 0.000, B 0.000, C 0.000 }
gfCNCPoint3[8346] = {X 353.2338, Y 102.6450, Z -3.8333, A 0.000, B 0.000, C 0.000 }
gfCNCPoint3[8347] = {X 347.7210, Y 102.7134, Z -3.8333, A 0.000, B 0.000, C 0.000 }
gfCNCPoint3[8348] = {X 342.2086, Y 102.6168, Z -3.8333, A 0.000, B 0.000, C 0.000 }
gfCNCPoint3[8349] = {X 336.7017, Y 102.3554, Z -3.8333, A 0.000, B 0.000, C 0.000 }
gfCNCPoint3[8350] = {X 333.2240, Y 102.0801, Z -3.8333, A 0.000, B 0.000, C 0.000 }
gfCNCPoint3[8351] = {X 329.7598, Y 101.6686, Z -3.8333, A 0.000, B 0.000, C 0.000 }
gfCNCPoint3[8352] = {X 326.3144, Y 101.1215, Z -3.8333, A 0.000, B 0.000, C 0.000 }
gfCNCPoint3[8353] = {X 323.4873, Y 100.5226, Z -3.8333, A 0.000, B 0.000, C 0.000 }
gfCNCPoint3[8354] = {X 320.7123, Y 99.7162, Z -3.8333, A 0.000, B 0.000, C 0.000 }
gfCNCPoint3[8355] = {X 318.0046, Y 98.7066, Z -3.8333, A 0.000, B 0.000, C 0.000 }
gfCNCPoint3[8356] = {X 316.5162, Y 98.0193, Z -3.8333, A 0.000, B 0.000, C 0.000 }
gfCNCPoint3[8357] = {X 315.0902, Y 97.2104, Z -3.8333, A 0.000, B 0.000, C 0.000 }
gfCNCPoint3[8358] = {X 313.7366, Y 96.2855, Z -3.8333, A 0.000, B 0.000, C 0.000 }
gfCNCPoint3[8359] = {X 312.4647, Y 95.2511, Z -3.8333, A 0.000, B 0.000, C 0.000 }
gfCNCPoint3[8360] = {X 311.4878, Y 94.2795, Z -3.8333, A 0.000, B 0.000, C 0.000 }
gfCNCPoint3[8361] = {X 310.6331, Y 93.1989, Z -3.8333, A 0.000, B 0.000, C 0.000 }
gfCNCPoint3[8362] = {X 309.9126, Y 92.0246, Z -3.8333, A 0.000, B 0.000, C 0.000 }
gfCNCPoint3[8363] = {X 309.3364, Y 90.7731, Z -3.8333, A 0.000, B 0.000, C 0.000 }
gfCNCPoint3[8364] = {X 308.9128, Y 89.4621, Z -3.8333, A 0.000, B 0.000, C 0.000 }
gfCNCPoint3[8365] = {X 308.5750, Y 87.8658, Z -3.8333, A 0.000, B 0.000, C 0.000 }
gfCNCPoint3[8366] = {X 308.3755, Y 86.2464, Z -3.8333, A 0.000, B 0.000, C 0.000 }
gfCNCPoint3[8367] = {X 308.3157, Y 84.6159, Z -3.8333, A 0.000, B 0.000, C 0.000 }
gfCNCPoint3[8368] = {X 308.3170, Y 62.9243, Z -3.8333, A 0.000, B 0.000, C 0.000 }
gfCNCPoint3[8369] = {X 307.4743, Y 62.7735, Z -3.8333, A 0.000, B 0.000, C 0.000 }
gfCNCPoint3[8370] = {X 306.6831, Y 62.4469, Z -3.8333, A 0.000, B 0.000, C 0.000 }
gfCNCPoint3[8371] = {X 305.9794, Y 61.9594, Z -3.8333, A 0.000, B 0.000, C 0.000 }
gfCNCPoint3[8372] = {X 305.3956, Y 61.3333, Z -3.8333, A 0.000, B 0.000, C 0.000 }
gfCNCPoint3[8373] = {X 304.9584, Y 60.5973, Z -3.8333, A 0.000, B 0.000, C 0.000 }
gfCNCPoint3[8374] = {X 304.6878, Y 59.7852, Z -3.8333, A 0.000, B 0.000, C 0.000 }
gfCNCPoint3[8375] = {X 304.5962, Y 58.9340, Z -3.8333, A 0.000, B 0.000, C 0.000 }
gfCNCPoint3[8376] = {X 304.5962, Y 58.0000, Z -3.8333, A 0.000, B 0.000, C 0.000 }
gfCNCPoint3[8377] = {X 304.6965, Y 57.1099, Z -3.8333, A 0.000, B 0.000, C 0.000 }
gfCNCPoint3[8378] = {X 304.9923, Y 56.2645, Z -3.8333, A 0.000, B 0.000, C 0.000 }
gfCNCPoint3[8379] = {X 305.4689, Y 55.5060, Z -3.8333, A 0.000, B 0.000, C 0.000 }
gfCNCPoint3[8380] = {X 306.1023, Y 54.8727, Z -3.8333, A 0.000, B 0.000, C 0.000 }
gfCNCPoint3[8381] = {X 306.8607, Y 54.3961, Z -3.8333, A 0.000, B 0.000, C 0.000 }
gfCNCPoint3[8382] = {X 307.7061, Y 54.1003, Z -3.8333, A 0.000, B 0.000, C 0.000 }
gfCNCPoint3[8383] = {X 308.5962, Y 54.0000, Z -3.8333, A 0.000, B 0.000, C 0.000 }
gfCNCPoint3[8384] = {X 324.3107, Y 54.0000, Z -3.8333, A 0.000, B 0.000, C 0.000 }
gfCNCPoint3[8385] = {X 325.2008, Y 54.1003, Z -3.8333, A 0.000, B 0.000, C 0.000 }
gfCNCPoint3[8386] = {X 326.0462, Y 54.3961, Z -3.8333, A 0.000, B 0.000, C 0.000 }
gfCNCPoint3[8387] = {X 326.8046, Y 54.8727, Z -3.8333, A 0.000, B 0.000, C 0.000 }
gfCNCPoint3[8388] = {X 327.4380, Y 55.5060, Z -3.8333, A 0.000, B 0.000, C 0.000 }
gfCNCPoint3[8389] = {X 327.9146, Y 56.2645, Z -3.8333, A 0.000, B 0.000, C 0.000 }
gfCNCPoint3[8390] = {X 328.2104, Y 57.1099, Z -3.8333, A 0.000, B 0.000, C 0.000 }
gfCNCPoint3[8391] = {X 328.3107, Y 58.0000, Z -3.8333, A 0.000, B 0.000, C 0.000 }
gfCNCPoint3[8392] = {X 328.3107, Y 58.9341, Z -3.8333, A 0.000, B 0.000, C 0.000 }
gfCNCPoint3[8393] = {X 328.2151, Y 59.7844, Z -3.8333, A 0.000, B 0.000, C 0.000 }
gfCNCPoint3[8394] = {X 327.9425, Y 60.5955, Z -3.8333, A 0.000, B 0.000, C 0.000 }
gfCNCPoint3[8395] = {X 327.5051, Y 61.3309, Z -3.8333, A 0.000, B 0.000, C 0.000 }
gfCNCPoint3[8396] = {X 326.9227, Y 61.9577, Z -3.8333, A 0.000, B 0.000, C 0.000 }
gfCNCPoint3[8397] = {X 326.2212, Y 62.4477, Z -3.8333, A 0.000, B 0.000, C 0.000 }
gfCNCPoint3[8398] = {X 325.4323, Y 62.7790, Z -3.8333, A 0.000, B 0.000, C 0.000 }
gfCNCPoint3[8399] = {X 324.5913, Y 62.9366, Z -3.8333, A 0.000, B 0.000, C 0.000 }
gfCNCPoint3[8400] = {X 324.5929, Y 83.2313, Z -3.8333, A 0.000, B 0.000, C 0.000 }
gfCNCPoint3[8401] = {X 324.6064, Y 84.6159, Z -3.8333, A 0.000, B 0.000, C 0.000 }
gfCNCPoint3[8402] = {X 324.6898, Y 85.9181, Z -3.8333, A 0.000, B 0.000, C 0.000 }
gfCNCPoint3[8403] = {X 324.9294, Y 87.2008, Z -3.8333, A 0.000, B 0.000, C 0.000 }
gfCNCPoint3[8404] = {X 325.2359, Y 87.5553, Z -3.8333, A 0.000, B 0.000, C 0.000 }
gfCNCPoint3[8405] = {X 325.6219, Y 87.8210, Z -3.8333, A 0.000, B 0.000, C 0.000 }
gfCNCPoint3[8406] = {X 326.0759, Y 88.0775, Z -3.8333, A 0.000, B 0.000, C 0.000 }
gfCNCPoint3[8407] = {X 327.5509, Y 88.6906, Z -3.8333, A 0.000, B 0.000, C 0.000 }
gfCNCPoint3[8408] = {X 329.0843, Y 89.1380, Z -3.8333, A 0.000, B 0.000, C 0.000 }
gfCNCPoint3[8409] = {X 332.1822, Y 89.7582, Z -3.8333, A 0.000, B 0.000, C 0.000 }
gfCNCPoint3[8410] = {X 335.3167, Y 90.1537, Z -3.8333, A 0.000, B 0.000, C 0.000 }
gfCNCPoint3[8411] = {X 339.4647, Y 90.4747, Z -3.8333, A 0.000, B 0.000, C 0.000 }
gfCNCPoint3[8412] = {X 343.6212, Y 90.6548, Z -3.8333, A 0.000, B 0.000, C 0.000 }
gfCNCPoint3[8413] = {X 347.7814, Y 90.6937, Z -3.8333, A 0.000, B 0.000, C 0.000 }
gfCNCPoint3[8414] = {X 352.1732, Y 90.6551, Z -3.8333, A 0.000, B 0.000, C 0.000 }
gfCNCPoint3[8415] = {X 356.5609, Y 90.4587, Z -3.8333, A 0.000, B 0.000, C 0.000 }
gfCNCPoint3[8416] = {X 360.9386, Y 90.1048, Z -3.8333, A 0.000, B 0.000, C 0.000 }
gfCNCPoint3[8417] = {X 363.2713, Y 89.8146, Z -3.8333, A 0.000, B 0.000, C 0.000 }
gfCNCPoint3[8418] = {X 365.5824, Y 89.3848, Z -3.8333, A 0.000, B 0.000, C 0.000 }
gfCNCPoint3[8419] = {X 367.8634, Y 88.8169, Z -3.8333, A 0.000, B 0.000, C 0.000 }
gfCNCPoint3[8420] = {X 368.8288, Y 88.4922, Z -3.8333, A 0.000, B 0.000, C 0.000 }
gfCNCPoint3[8421] = {X 369.7518, Y 88.0613, Z -3.8333, A 0.000, B 0.000, C 0.000 }
gfCNCPoint3[8422] = {X 370.6206, Y 87.5297, Z -3.8333, A 0.000, B 0.000, C 0.000 }
gfCNCPoint3[8423] = {X 370.8585, Y 87.2820, Z -3.8333, A 0.000, B 0.000, C 0.000 }
gfCNCPoint3[8424] = {X 370.9812, Y 86.9612, Z -3.8333, A 0.000, B 0.000, C 0.000 }
gfCNCPoint3[8425] = {X 371.1756, Y 85.4000, Z -3.8333, A 0.000, B 0.000, C 0.000 }
gfCNCPoint3[8426] = {X 371.2404, Y 83.8281, Z -3.8333, A 0.000, B 0.000, C 0.000 }
gfCNCPoint3[8427] = {X 371.2389, Y 63.0390, Z -3.8333, A 0.000, B 0.000, C 0.000 }
gfCNCPoint3[8428] = {X 371.2440, Y 62.9246, Z -3.8333, A 0.000, B 0.000, C 0.000 }
gfCNCPoint3[8429] = {X 371.0720, Y 62.9090, Z -3.8333, A 0.000, B 0.000, C 0.000 }
gfCNCPoint3[8430] = {X 370.9007, Y 62.8860, Z -3.8333, A 0.000, B 0.000, C 0.000 }
gfCNCPoint3[8431] = {X 369.9942, Y 62.6319, Z -3.8333, A 0.000, B 0.000, C 0.000 }
gfCNCPoint3[8432] = {X 369.1721, Y 62.1730, Z -3.8333, A 0.000, B 0.000, C 0.000 }
gfCNCPoint3[8433] = {X 368.4800, Y 61.5346, Z -3.8333, A 0.000, B 0.000, C 0.000 }
gfCNCPoint3[8434] = {X 367.9564, Y 60.7522, Z -3.8333, A 0.000, B 0.000, C 0.000 }
gfCNCPoint3[8435] = {X 367.6301, Y 59.8690, Z -3.8333, A 0.000, B 0.000, C 0.000 }
gfCNCPoint3[8436] = {X 367.5193, Y 58.9340, Z -3.8333, A 0.000, B 0.000, C 0.000 }
gfCNCPoint3[8437] = {X 367.5193, Y 58.0000, Z -3.8333, A 0.000, B 0.000, C 0.000 }
gfCNCPoint3[8438] = {X 367.6196, Y 57.1099, Z -3.8333, A 0.000, B 0.000, C 0.000 }
gfCNCPoint3[8439] = {X 367.9154, Y 56.2645, Z -3.8333, A 0.000, B 0.000, C 0.000 }
gfCNCPoint3[8440] = {X 368.3920, Y 55.5060, Z -3.8333, A 0.000, B 0.000, C 0.000 }
gfCNCPoint3[8441] = {X 369.0253, Y 54.8727, Z -3.8333, A 0.000, B 0.000, C 0.000 }
gfCNCPoint3[8442] = {X 369.7837, Y 54.3961, Z -3.8333, A 0.000, B 0.000, C 0.000 }
gfCNCPoint3[8443] = {X 370.6292, Y 54.1003, Z -3.8333, A 0.000, B 0.000, C 0.000 }
gfCNCPoint3[8444] = {X 371.5193, Y 54.0000, Z -3.8333, A 0.000, B 0.000, C 0.000 }
gfCNCPoint3[8445] = {X 388.0597, Y 54.0000, Z -3.8333, A 0.000, B 0.000, C 0.000 }
gfCNCPoint3[8446] = {X 388.9498, Y 54.1003, Z -3.8333, A 0.000, B 0.000, C 0.000 }
gfCNCPoint3[8447] = {X 389.7952, Y 54.3961, Z -3.8333, A 0.000, B 0.000, C 0.000 }
gfCNCPoint3[8448] = {X 390.5536, Y 54.8727, Z -3.8333, A 0.000, B 0.000, C 0.000 }
gfCNCPoint3[8449] = {X 391.1870, Y 55.5060, Z -3.8333, A 0.000, B 0.000, C 0.000 }
gfCNCPoint3[8450] = {X 391.6636, Y 56.2645, Z -3.8333, A 0.000, B 0.000, C 0.000 }
gfCNCPoint3[8451] = {X 391.9594, Y 57.1099, Z -3.8333, A 0.000, B 0.000, C 0.000 }
gfCNCPoint3[8452] = {X 392.0597, Y 58.0000, Z -3.8333, A 0.000, B 0.000, C 0.000 }
gfCNCPoint3[8453] = {X 392.0595, Y 58.9671, Z -3.8333, A 0.000, B 0.000, C 0.000 }
gfCNCPoint3[8454] = {X 391.9499, Y 59.8647, Z -3.8333, A 0.000, B 0.000, C 0.000 }
gfCNCPoint3[8455] = {X 391.6414, Y 60.7148, Z -3.8333, A 0.000, B 0.000, C 0.000 }
gfCNCPoint3[8456] = {X 391.1186, Y 61.5124, Z -3.8333, A 0.000, B 0.000, C 0.000 }
gfCNCPoint3[8457] = {X 390.4226, Y 62.1645, Z -3.8333, A 0.000, B 0.000, C 0.000 }
gfCNCPoint3[8458] = {X 389.5927, Y 62.6344, Z -3.8333, A 0.000, B 0.000, C 0.000 }
gfCNCPoint3[8459] = {X 388.6754, Y 62.8957, Z -3.8333, A 0.000, B 0.000, C 0.000 }
gfCNCPoint3[8460] = {X 388.5093, Y 62.9187, Z -3.8333, A 0.000, B 0.000, C 0.000 }
gfCNCPoint3[8461] = {X 388.3422, Y 62.9348, Z -3.8333, A 0.000, B 0.000, C 0.000 }
gfCNCPoint3[8462] = {X 388.3386, Y 63.1540, Z -3.8333, A 0.000, B 0.000, C 0.000 }
gfCNCPoint3[8463] = {X 388.3386, Y 83.9236, Z -3.8333, A 0.000, B 0.000, C 0.000 }
gfCNCPoint3[8464] = {X 388.3366, Y 84.6159, Z -3.8333, A 0.000, B 0.000, C 0.000 }
gfCNCPoint3[8465] = {X 388.2778, Y 86.2468, Z -3.8333, A 0.000, B 0.000, C 0.000 }
gfCNCPoint3[8466] = {X 388.0769, Y 87.8663, Z -3.8333, A 0.000, B 0.000, C 0.000 }
gfCNCPoint3[8467] = {X 387.7354, Y 89.4621, Z -3.8333, A 0.000, B 0.000, C 0.000 }
gfCNCPoint3[8468] = {X 387.2176, Y 91.0069, Z -3.8333, A 0.000, B 0.000, C 0.000 }
gfCNCPoint3[8469] = {X 386.4882, Y 92.4637, Z -3.8333, A 0.000, B 0.000, C 0.000 }
gfCNCPoint3[8470] = {X 385.5616, Y 93.8038, Z -3.8333, A 0.000, B 0.000, C 0.000 }
gfCNCPoint3[8471] = {X 384.4563, Y 95.0007, Z -3.8333, A 0.000, B 0.000, C 0.000 }
gfCNCPoint3[8472] = {X 382.9680, Y 96.2546, Z -3.8333, A 0.000, B 0.000, C 0.000 }
gfCNCPoint3[8473] = {X 381.3551, Y 97.3434, Z -3.8333, A 0.000, B 0.000, C 0.000 }
